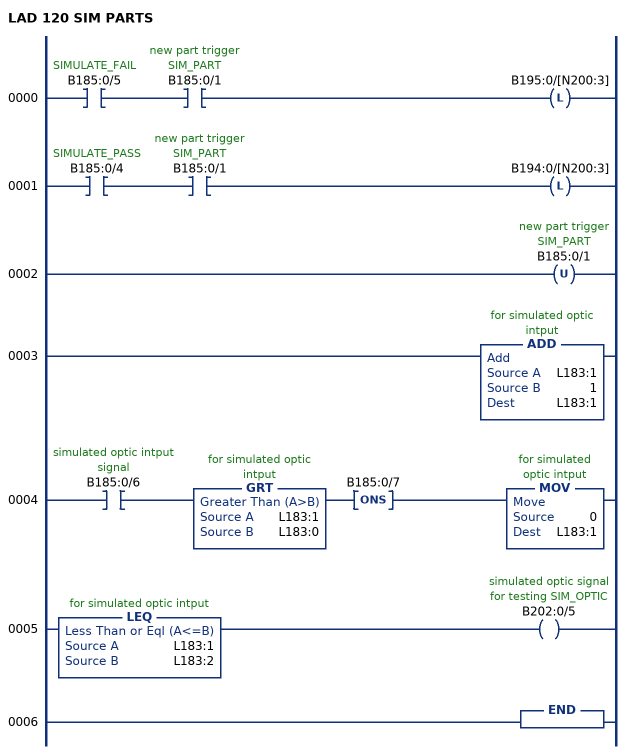
% Rung: 0 %
SOR XIC B185:0/5 XIC B185:0/1 OTL B195:0/[N200:3] EOR
%   B185:0/5  SIMULATE_FAIL %
%   B185:0/1  SIM_PART  "new part trigger" %
%   N200:3  OPT_LD_PT %
% Rung: 1 %
SOR XIC B185:0/4 XIC B185:0/1 OTL B194:0/[N200:3] EOR
%   B185:0/4  SIMULATE_PASS %
%   B185:0/1  SIM_PART  "new part trigger" %
%   N200:3  OPT_LD_PT %
% Rung: 2 %
SOR OTU B185:0/1 EOR
%   B185:0/1  SIM_PART  "new part trigger" %
% Rung: 3 %
SOR ADD L183:1 1 L183:1 EOR
%   L183:1  "for simulated optic intput" %
% Rung: 4 %
SOR XIC B185:0/6 GRT L183:1 L183:0 ONS B185:0/7 MOV 0 L183:1 EOR
%   B185:0/6  "simulated optic intput signal" %
%   L183:1  "for simulated optic intput" %
%   L183:0  "count for part data injection" %
% Rung: 5 %
SOR LEQ L183:1 L183:2 OTE B202:0/5 EOR
%   L183:1  "for simulated optic intput" %
%   L183:2  "simulated part width" %
%   B202:0/5  SIM_OPTIC  "simulated optic signal for testing" %
% Rung: 6 %
SOR END EOR

LADDER 121 "PARTDETECT"
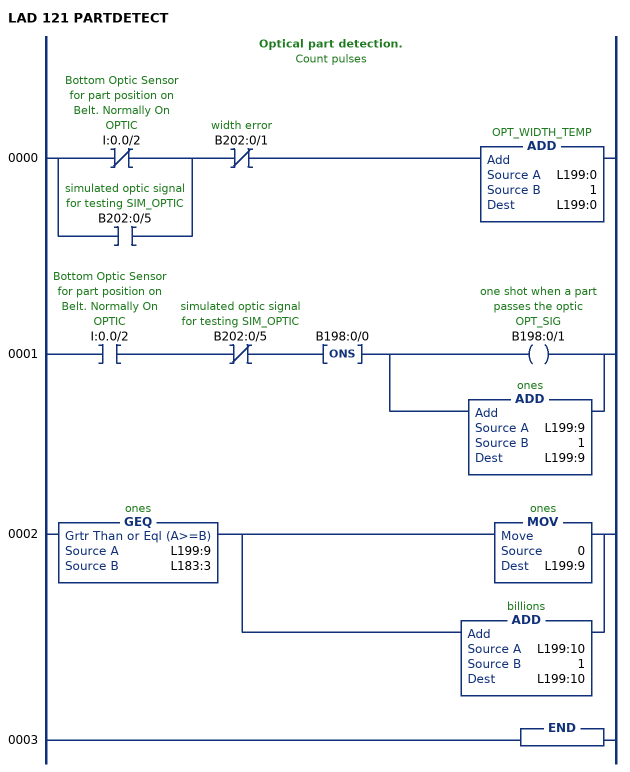
% Rung: 0 %
% TITLE: Optical part detection. %
% Count pulses %
SOR BST XIO I:0.0/2 NXB XIC B202:0/5 BND XIO B202:0/1 ADD L199:0 1 L199:0 EOR
%   I:0.0/2  OPTIC  "Bottom Optic Sensor for part position on Belt. Normally On" %
%   B202:0/5  SIM_OPTIC  "simulated optic signal for testing" %
%   B202:0/1  "width error" %
%   L199:0  OPT_WIDTH_TEMP %
% Rung: 1 %
SOR XIC I:0.0/2 XIO B202:0/5 ONS B198:0/0 BST OTE B198:0/1 NXB ADD L199:9 1 L199:9 BND EOR
%   I:0.0/2  OPTIC  "Bottom Optic Sensor for part position on Belt. Normally On" %
%   B202:0/5  SIM_OPTIC  "simulated optic signal for testing" %
%   B198:0/1  OPT_SIG  "one shot when a part passes the optic" %
%   L199:9  "ones" %
% Rung: 2 %
SOR GEQ L199:9 L183:3 BST MOV 0 L199:9 NXB ADD L199:10 1 L199:10 BND EOR
%   L199:9  "ones" %
%   L183:3  "button state" %
%   L199:10  "billions" %
% Rung: 3 %
SOR END EOR

LADDER 122 "OPTICWIDTH"
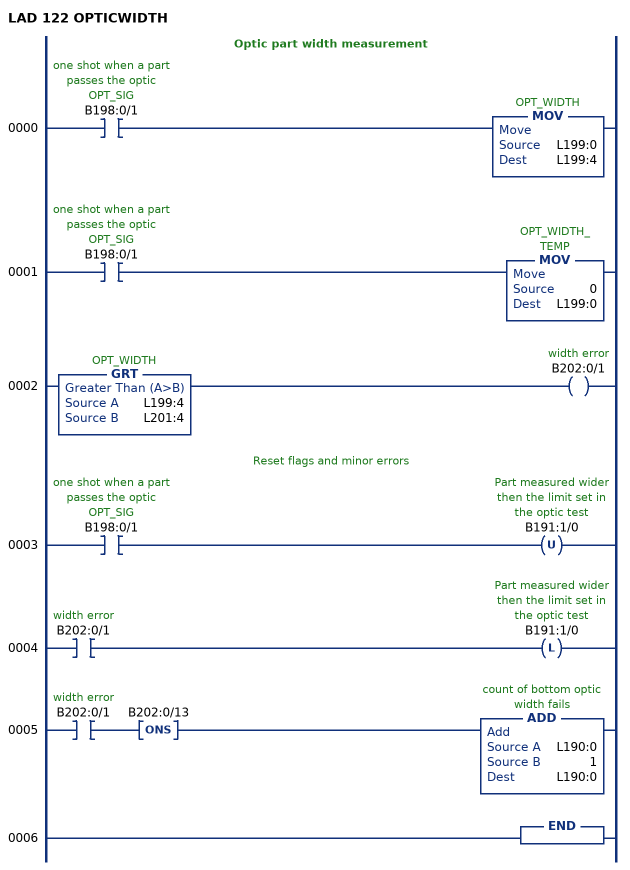
% Rung: 0 %
% TITLE: Optic part width measurement %
SOR XIC B198:0/1 MOV L199:0 L199:4 EOR
%   B198:0/1  OPT_SIG  "one shot when a part passes the optic" %
%   L199:0  OPT_WIDTH_TEMP %
%   L199:4  OPT_WIDTH %
% Rung: 1 %
SOR XIC B198:0/1 MOV 0 L199:0 EOR
%   B198:0/1  OPT_SIG  "one shot when a part passes the optic" %
%   L199:0  OPT_WIDTH_TEMP %
% Rung: 2 %
SOR GRT L199:4 L201:4 OTE B202:0/1 EOR
%   L199:4  OPT_WIDTH %
%   L201:4  MAX_WIDTH  "hmi in" %
%   B202:0/1  "width error" %
% Rung: 3 %
% Reset flags and minor errors %
SOR XIC B198:0/1 OTU B191:1/0 EOR
%   B198:0/1  OPT_SIG  "one shot when a part passes the optic" %
%   B191:1/0  "Part measured wider then the limit set in the optic test" %
% Rung: 4 %
SOR XIC B202:0/1 OTL B191:1/0 EOR
%   B202:0/1  "width error" %
%   B191:1/0  "Part measured wider then the limit set in the optic test" %
% Rung: 5 %
SOR XIC B202:0/1 ONS B202:0/13 ADD L190:0 1 L190:0 EOR
%   B202:0/1  "width error" %
%   L190:0  "count of bottom optic width fails" %
% Rung: 6 %
SOR END EOR

LADDER 123 "PART GAP"
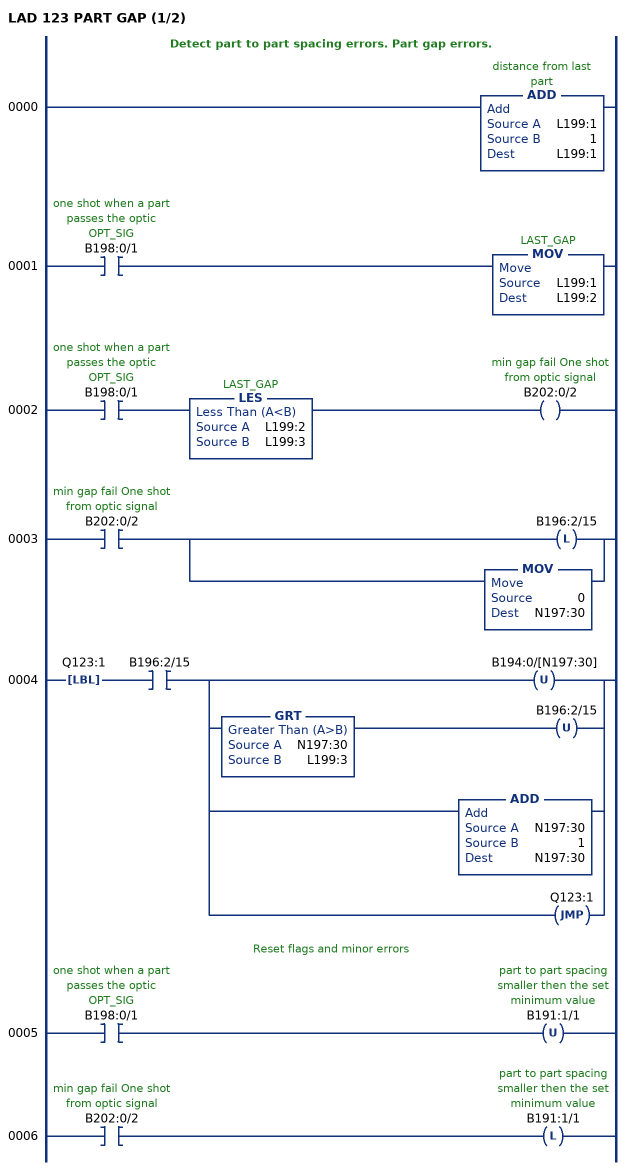
% Rung: 0 %
% TITLE: Detect part to part spacing errors. Part gap errors. %
SOR ADD L199:1 1 L199:1 EOR
%   L199:1  "distance from last part" %
% Rung: 1 %
SOR XIC B198:0/1 MOV L199:1 L199:2 EOR
%   B198:0/1  OPT_SIG  "one shot when a part passes the optic" %
%   L199:1  "distance from last part" %
%   L199:2  LAST_GAP %
% Rung: 2 %
SOR XIC B198:0/1 LES L199:2 L199:3 OTE B202:0/2 EOR
%   B198:0/1  OPT_SIG  "one shot when a part passes the optic" %
%   L199:2  LAST_GAP %
%   L199:3  MIN_WIDTH %
%   B202:0/2  "min gap fail One shot from optic signal" %
% Rung: 3 %
SOR XIC B202:0/2 BST OTL B196:2/15 NXB MOV 0 N197:30 BND EOR
%   B202:0/2  "min gap fail One shot from optic signal" %
% Rung: 4 %
SOR LBL Q123:1 XIC B196:2/15 BST OTU B194:0/[N197:30] NXB GRT N197:30 L199:3 OTU B196:2/15 NXB ADD N197:30 1 N197:30 NXB JMP Q123:1 BND EOR
%   L199:3  MIN_WIDTH %
% Rung: 5 %
% Reset flags and minor errors %
SOR XIC B198:0/1 OTU B191:1/1 EOR
%   B198:0/1  OPT_SIG  "one shot when a part passes the optic" %
%   B191:1/1  "part to part spacing smaller then the set minimum value" %
% Rung: 6 %
SOR XIC B202:0/2 OTL B191:1/1 EOR
%   B202:0/2  "min gap fail One shot from optic signal" %
%   B191:1/1  "part to part spacing smaller then the set minimum value" %

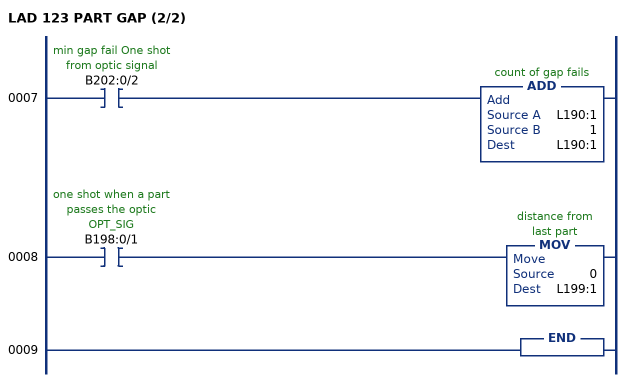
% Rung: 7 %
SOR XIC B202:0/2 ADD L190:1 1 L190:1 EOR
%   B202:0/2  "min gap fail One shot from optic signal" %
%   L190:1  "count of gap fails" %
% Rung: 8 %
SOR XIC B198:0/1 MOV 0 L199:1 EOR
%   B198:0/1  OPT_SIG  "one shot when a part passes the optic" %
%   L199:1  "distance from last part" %
% Rung: 9 %
SOR END EOR

LADDER 125 "OPTIC"
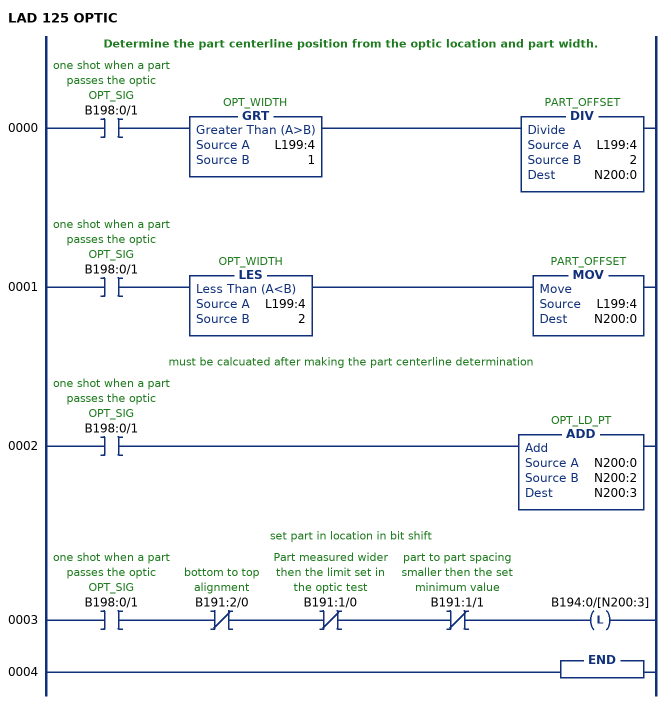
% Rung: 0 %
% TITLE: Determine the part centerline position from the optic location and part width. %
SOR XIC B198:0/1 GRT L199:4 1 DIV L199:4 2 N200:0 EOR
%   B198:0/1  OPT_SIG  "one shot when a part passes the optic" %
%   L199:4  OPT_WIDTH %
%   N200:0  PART_OFFSET %
% Rung: 1 %
SOR XIC B198:0/1 LES L199:4 2 MOV L199:4 N200:0 EOR
%   B198:0/1  OPT_SIG  "one shot when a part passes the optic" %
%   L199:4  OPT_WIDTH %
%   N200:0  PART_OFFSET %
% Rung: 2 %
% must be calcuated after making the part centerline determination %
SOR XIC B198:0/1 ADD N200:0 N200:2 N200:3 EOR
%   B198:0/1  OPT_SIG  "one shot when a part passes the optic" %
%   N200:0  PART_OFFSET %
%   N200:2  OPTIC_LOC %
%   N200:3  OPT_LD_PT %
% Rung: 3 %
% set part in location in bit shift %
SOR XIC B198:0/1 XIO B191:2/0 XIO B191:1/0 XIO B191:1/1 OTL B194:0/[N200:3] EOR
%   B198:0/1  OPT_SIG  "one shot when a part passes the optic" %
%   B191:2/0  "bottom to top alignment" %
%   B191:1/0  "Part measured wider then the limit set in the optic test" %
%   B191:1/1  "part to part spacing smaller then the set minimum value" %
%   N200:3  OPT_LD_PT %
% Rung: 4 %
SOR END EOR

LADDER 130 "INS 1 TRIG"
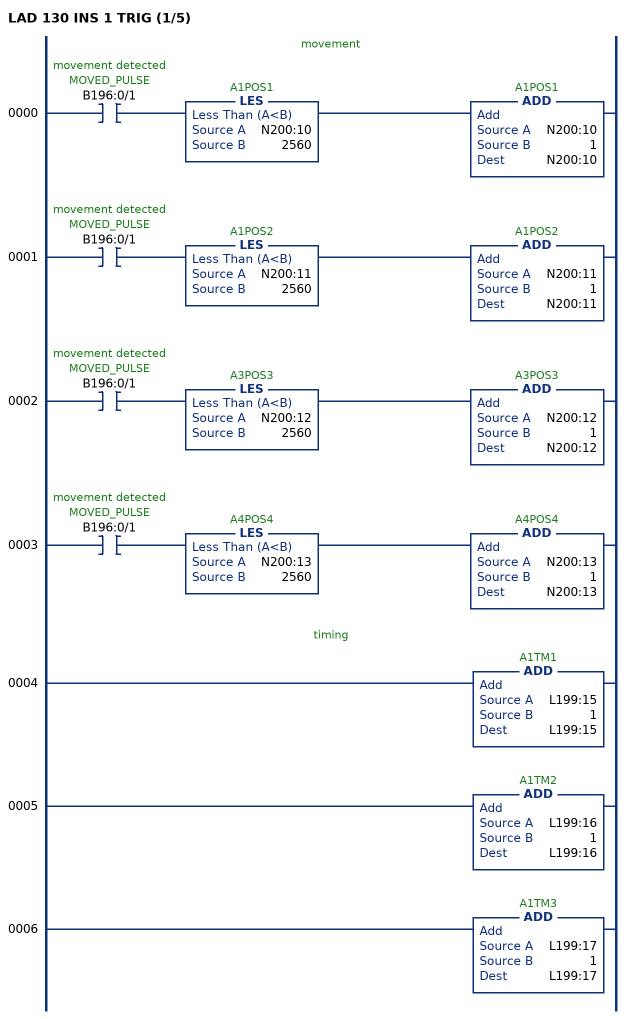
% Rung: 0 %
% movement %
SOR XIC B196:0/1 LES N200:10 2560 ADD N200:10 1 N200:10 EOR
%   B196:0/1  MOVED_PULSE  "movement detected" %
%   N200:10  A1POS1 %
% Rung: 1 %
SOR XIC B196:0/1 LES N200:11 2560 ADD N200:11 1 N200:11 EOR
%   B196:0/1  MOVED_PULSE  "movement detected" %
%   N200:11  A1POS2 %
% Rung: 2 %
SOR XIC B196:0/1 LES N200:12 2560 ADD N200:12 1 N200:12 EOR
%   B196:0/1  MOVED_PULSE  "movement detected" %
%   N200:12  A3POS3 %
% Rung: 3 %
SOR XIC B196:0/1 LES N200:13 2560 ADD N200:13 1 N200:13 EOR
%   B196:0/1  MOVED_PULSE  "movement detected" %
%   N200:13  A4POS4 %
% Rung: 4 %
% timing %
SOR ADD L199:15 1 L199:15 EOR
%   L199:15  A1TM1 %
% Rung: 5 %
SOR ADD L199:16 1 L199:16 EOR
%   L199:16  A1TM2 %
% Rung: 6 %
SOR ADD L199:17 1 L199:17 EOR
%   L199:17  A1TM3 %

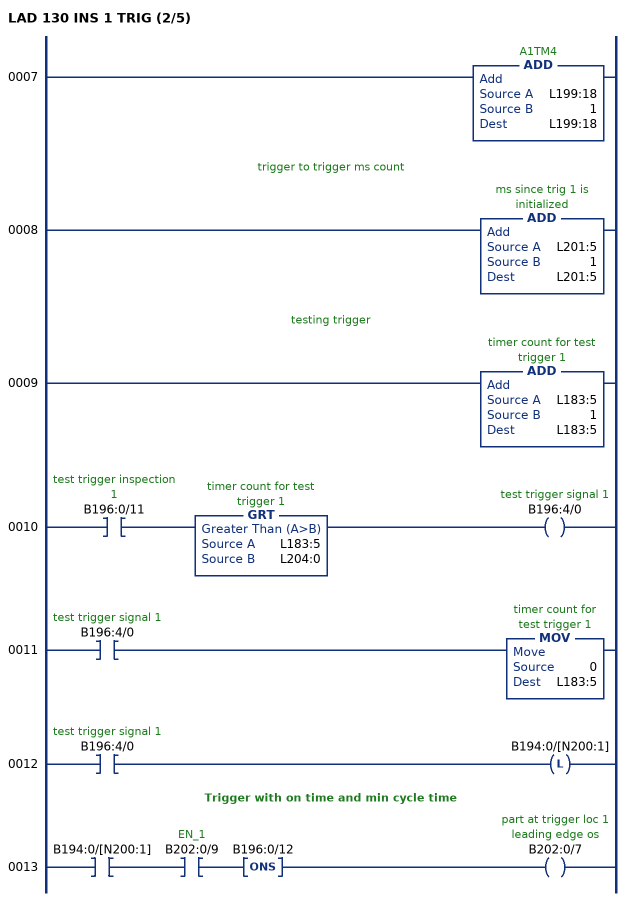
% Rung: 7 %
SOR ADD L199:18 1 L199:18 EOR
%   L199:18  A1TM4 %
% Rung: 8 %
% trigger to trigger ms count %
SOR ADD L201:5 1 L201:5 EOR
%   L201:5  "ms since trig 1 is initialized" %
% Rung: 9 %
% testing trigger %
SOR ADD L183:5 1 L183:5 EOR
%   L183:5  "timer count for test trigger 1" %
% Rung: 10 %
SOR XIC B196:0/11 GRT L183:5 L204:0 OTE B196:4/0 EOR
%   B196:0/11  "test trigger inspection 1" %
%   L183:5  "timer count for test trigger 1" %
%   B196:4/0  "test trigger signal 1" %
% Rung: 11 %
SOR XIC B196:4/0 MOV 0 L183:5 EOR
%   B196:4/0  "test trigger signal 1" %
%   L183:5  "timer count for test trigger 1" %
% Rung: 12 %
SOR XIC B196:4/0 OTL B194:0/[N200:1] EOR
%   B196:4/0  "test trigger signal 1" %
%   N200:1  INS_1_TRIG_LOC %
% Rung: 13 %
% TITLE: Trigger with on time and min cycle time %
SOR XIC B194:0/[N200:1] XIC B202:0/9 ONS B196:0/12 OTE B202:0/7 EOR
%   N200:1  INS_1_TRIG_LOC %
%   B202:0/9  EN_1 %
%   B202:0/7  "part at trigger loc 1 leading edge os" %

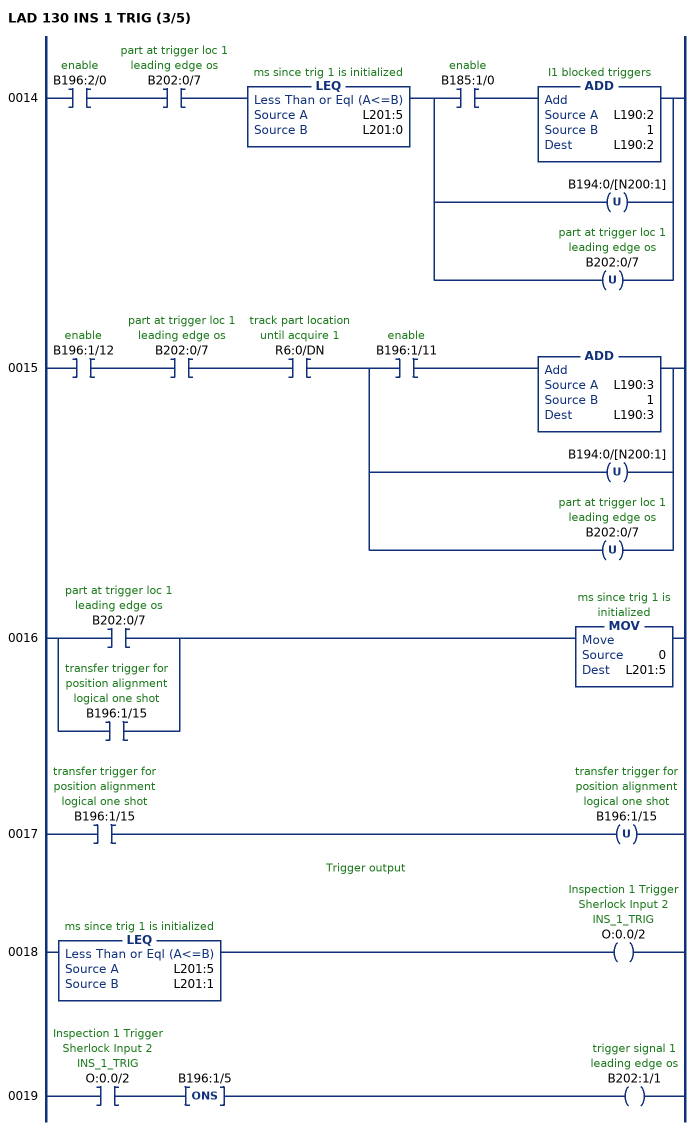
% Rung: 14 %
SOR XIC B196:2/0 XIC B202:0/7 LEQ L201:5 L201:0 BST XIC B185:1/0 ADD L190:2 1 L190:2 NXB OTU B194:0/[N200:1] NXB OTU B202:0/7 BND EOR
%   B196:2/0  "enable" %
%   B202:0/7  "part at trigger loc 1 leading edge os" %
%   L201:5  "ms since trig 1 is initialized" %
%   L201:0  CAM_1_MIN_CYCLE_TIME %
%   B185:1/0  "enable" %
%   L190:2  "I1 blocked triggers" %
%   N200:1  INS_1_TRIG_LOC %
% Rung: 15 %
SOR XIC B196:1/12 XIC B202:0/7 XIC R6:0/DN BST XIC B196:1/11 ADD L190:3 1 L190:3 NXB OTU B194:0/[N200:1] NXB OTU B202:0/7 BND EOR
%   B196:1/12  "enable" %
%   B202:0/7  "part at trigger loc 1 leading edge os" %
%   R6:0  "track part location until acquire 1" %
%   B196:1/11  "enable" %
%   N200:1  INS_1_TRIG_LOC %
% Rung: 16 %
SOR BST XIC B202:0/7 NXB XIC B196:1/15 BND MOV 0 L201:5 EOR
%   B202:0/7  "part at trigger loc 1 leading edge os" %
%   B196:1/15  "transfer trigger for position alignment logical one shot" %
%   L201:5  "ms since trig 1 is initialized" %
% Rung: 17 %
SOR XIC B196:1/15 OTU B196:1/15 EOR
%   B196:1/15  "transfer trigger for position alignment logical one shot" %
% Rung: 18 %
% Trigger output %
SOR LEQ L201:5 L201:1 OTE O:0.0/2 EOR
%   L201:5  "ms since trig 1 is initialized" %
%   L201:1  CAM_1_TRIG_TIME  "out time" %
%   O:0.0/2  INS_1_TRIG  "Inspection 1 Trigger Sherlock Input 2" %
% Rung: 19 %
SOR XIC O:0.0/2 ONS B196:1/5 OTE B202:1/1 EOR
%   O:0.0/2  INS_1_TRIG  "Inspection 1 Trigger Sherlock Input 2" %
%   B202:1/1  "trigger signal 1 leading edge os" %

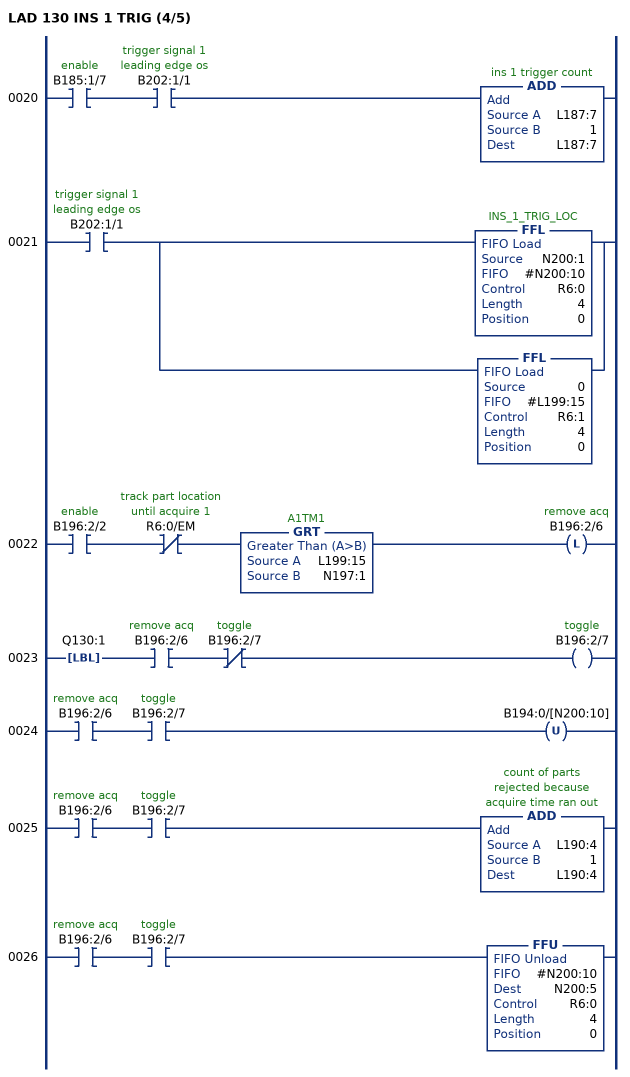
% Rung: 20 %
SOR XIC B185:1/7 XIC B202:1/1 ADD L187:7 1 L187:7 EOR
%   B185:1/7  "enable" %
%   B202:1/1  "trigger signal 1 leading edge os" %
%   L187:7  "ins 1 trigger count" %
% Rung: 21 %
SOR XIC B202:1/1 BST FFL N200:1 #N200:10 R6:0 4 0 NXB FFL 0 #L199:15 R6:1 4 0 BND EOR
%   B202:1/1  "trigger signal 1 leading edge os" %
%   N200:1  INS_1_TRIG_LOC %
%   N200:10  A1POS1 %
%   R6:0  "track part location until acquire 1" %
%   L199:15  A1TM1 %
%   R6:1  "track acquire time 1" %
% Rung: 22 %
SOR XIC B196:2/2 XIO R6:0/EM GRT L199:15 N197:1 OTL B196:2/6 EOR
%   B196:2/2  "enable" %
%   R6:0  "track part location until acquire 1" %
%   L199:15  A1TM1 %
%   N197:1  "maximim acquire time 1" %
%   B196:2/6  "remove acq" %
% Rung: 23 %
SOR LBL Q130:1 XIC B196:2/6 XIO B196:2/7 OTE B196:2/7 EOR
%   B196:2/6  "remove acq" %
%   B196:2/7  "toggle" %
% Rung: 24 %
SOR XIC B196:2/6 XIC B196:2/7 OTU B194:0/[N200:10] EOR
%   B196:2/6  "remove acq" %
%   B196:2/7  "toggle" %
%   N200:10  A1POS1 %
% Rung: 25 %
SOR XIC B196:2/6 XIC B196:2/7 ADD L190:4 1 L190:4 EOR
%   B196:2/6  "remove acq" %
%   B196:2/7  "toggle" %
%   L190:4  "count of parts rejected because acquire time ran out" %
% Rung: 26 %
SOR XIC B196:2/6 XIC B196:2/7 FFU #N200:10 N200:5 R6:0 4 0 EOR
%   B196:2/6  "remove acq" %
%   B196:2/7  "toggle" %
%   N200:10  A1POS1 %
%   R6:0  "track part location until acquire 1" %

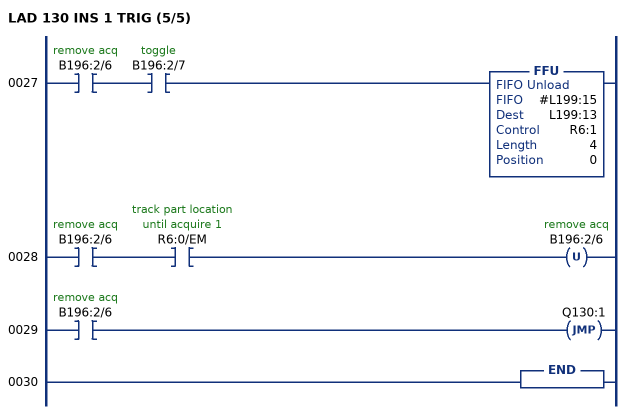
% Rung: 27 %
SOR XIC B196:2/6 XIC B196:2/7 FFU #L199:15 L199:13 R6:1 4 0 EOR
%   B196:2/6  "remove acq" %
%   B196:2/7  "toggle" %
%   L199:15  A1TM1 %
%   R6:1  "track acquire time 1" %
% Rung: 28 %
SOR XIC B196:2/6 XIC R6:0/EM OTU B196:2/6 EOR
%   B196:2/6  "remove acq" %
%   R6:0  "track part location until acquire 1" %
% Rung: 29 %
SOR XIC B196:2/6 JMP Q130:1 EOR
%   B196:2/6  "remove acq" %
% Rung: 30 %
SOR END EOR

LADDER 131 "INS 1 RSLT"
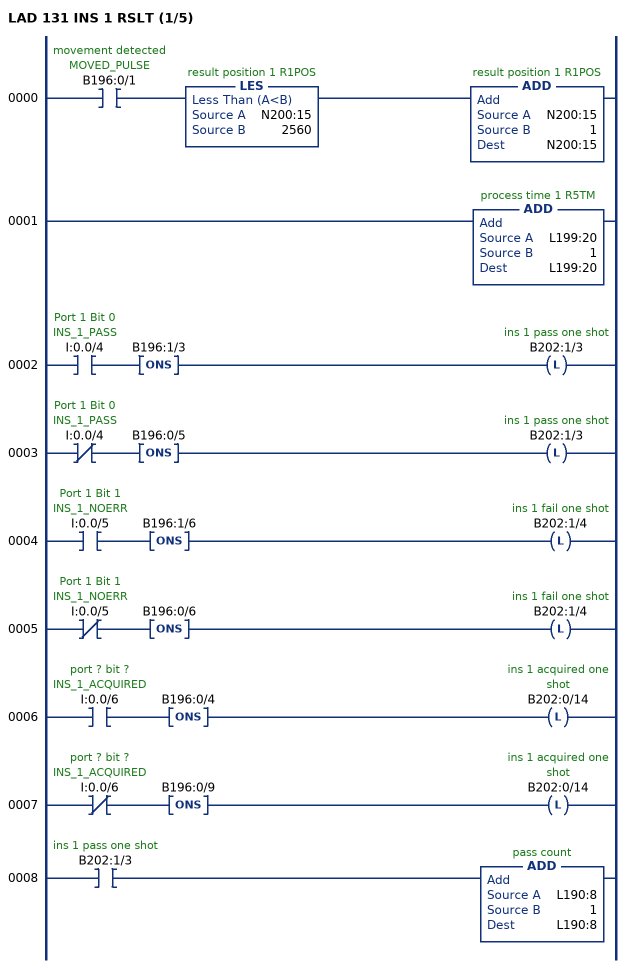
% Rung: 0 %
SOR XIC B196:0/1 LES N200:15 2560 ADD N200:15 1 N200:15 EOR
%   B196:0/1  MOVED_PULSE  "movement detected" %
%   N200:15  R1POS  "result position 1" %
% Rung: 1 %
SOR ADD L199:20 1 L199:20 EOR
%   L199:20  R5TM  "process time 1" %
% Rung: 2 %
SOR XIC I:0.0/4 ONS B196:1/3 OTL B202:1/3 EOR
%   I:0.0/4  INS_1_PASS  "Port 1 Bit 0" %
%   B202:1/3  "ins 1 pass one shot" %
% Rung: 3 %
SOR XIO I:0.0/4 ONS B196:0/5 OTL B202:1/3 EOR
%   I:0.0/4  INS_1_PASS  "Port 1 Bit 0" %
%   B202:1/3  "ins 1 pass one shot" %
% Rung: 4 %
SOR XIC I:0.0/5 ONS B196:1/6 OTL B202:1/4 EOR
%   I:0.0/5  INS_1_NOERR  "Port 1 Bit 1" %
%   B202:1/4  "ins 1 fail one shot" %
% Rung: 5 %
SOR XIO I:0.0/5 ONS B196:0/6 OTL B202:1/4 EOR
%   I:0.0/5  INS_1_NOERR  "Port 1 Bit 1" %
%   B202:1/4  "ins 1 fail one shot" %
% Rung: 6 %
SOR XIC I:0.0/6 ONS B196:0/4 OTL B202:0/14 EOR
%   I:0.0/6  INS_1_ACQUIRED  "port ? bit ?" %
%   B202:0/14  "ins 1 acquired one shot" %
% Rung: 7 %
SOR XIO I:0.0/6 ONS B196:0/9 OTL B202:0/14 EOR
%   I:0.0/6  INS_1_ACQUIRED  "port ? bit ?" %
%   B202:0/14  "ins 1 acquired one shot" %
% Rung: 8 %
SOR XIC B202:1/3 ADD L190:8 1 L190:8 EOR
%   B202:1/3  "ins 1 pass one shot" %
%   L190:8  "pass count" %

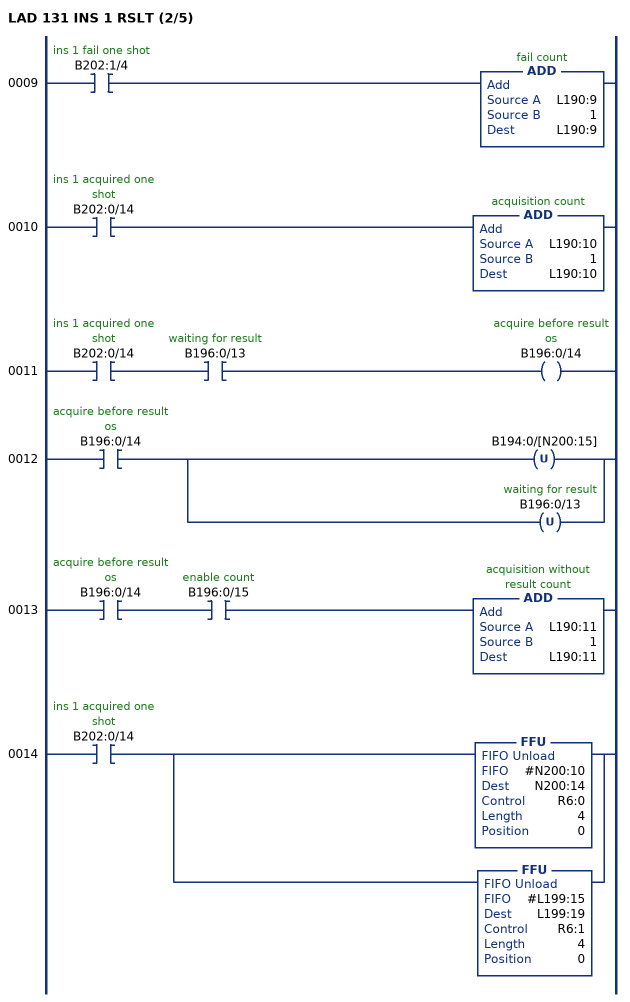
% Rung: 9 %
SOR XIC B202:1/4 ADD L190:9 1 L190:9 EOR
%   B202:1/4  "ins 1 fail one shot" %
%   L190:9  "fail count" %
% Rung: 10 %
SOR XIC B202:0/14 ADD L190:10 1 L190:10 EOR
%   B202:0/14  "ins 1 acquired one shot" %
%   L190:10  "acquisition count" %
% Rung: 11 %
SOR XIC B202:0/14 XIC B196:0/13 OTE B196:0/14 EOR
%   B202:0/14  "ins 1 acquired one shot" %
%   B196:0/13  "waiting for result" %
%   B196:0/14  "acquire before result os" %
% Rung: 12 %
SOR XIC B196:0/14 BST OTU B194:0/[N200:15] NXB OTU B196:0/13 BND EOR
%   B196:0/14  "acquire before result os" %
%   N200:15  R1POS  "result position 1" %
%   B196:0/13  "waiting for result" %
% Rung: 13 %
SOR XIC B196:0/14 XIC B196:0/15 ADD L190:11 1 L190:11 EOR
%   B196:0/14  "acquire before result os" %
%   B196:0/15  "enable count" %
%   L190:11  "acquisition without result count" %
% Rung: 14 %
SOR XIC B202:0/14 BST FFU #N200:10 N200:14 R6:0 4 0 NXB FFU #L199:15 L199:19 R6:1 4 0 BND EOR
%   B202:0/14  "ins 1 acquired one shot" %
%   N200:10  A1POS1 %
%   R6:0  "track part location until acquire 1" %
%   L199:15  A1TM1 %
%   R6:1  "track acquire time 1" %

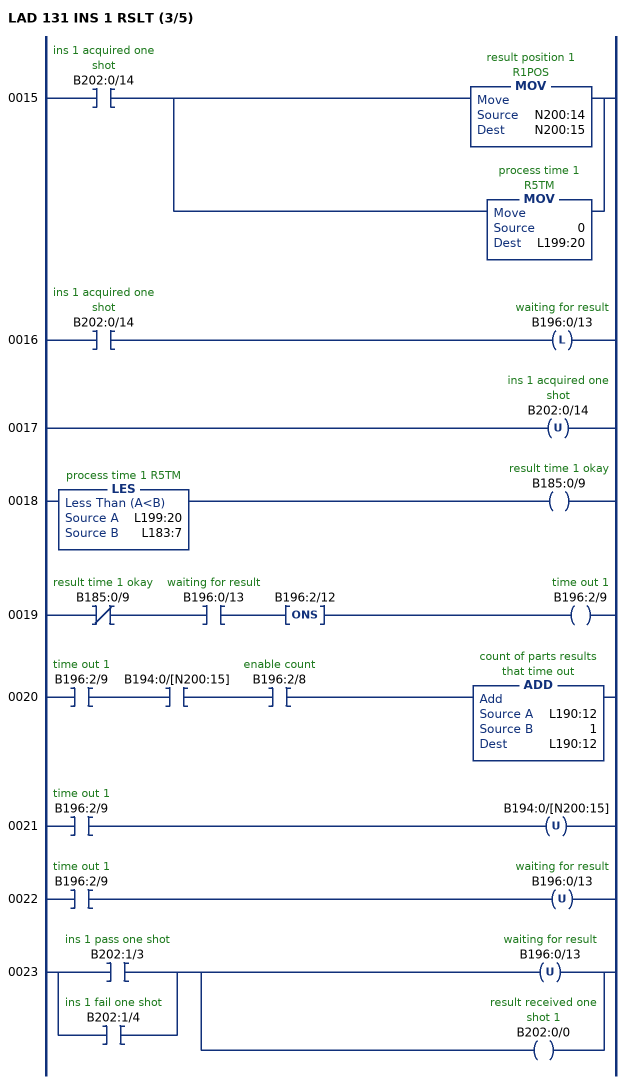
% Rung: 15 %
SOR XIC B202:0/14 BST MOV N200:14 N200:15 NXB MOV 0 L199:20 BND EOR
%   B202:0/14  "ins 1 acquired one shot" %
%   N200:15  R1POS  "result position 1" %
%   L199:20  R5TM  "process time 1" %
% Rung: 16 %
SOR XIC B202:0/14 OTL B196:0/13 EOR
%   B202:0/14  "ins 1 acquired one shot" %
%   B196:0/13  "waiting for result" %
% Rung: 17 %
SOR OTU B202:0/14 EOR
%   B202:0/14  "ins 1 acquired one shot" %
% Rung: 18 %
SOR LES L199:20 L183:7 OTE B185:0/9 EOR
%   L199:20  R5TM  "process time 1" %
%   L183:7  "max process time 1" %
%   B185:0/9  "result time 1 okay" %
% Rung: 19 %
SOR XIO B185:0/9 XIC B196:0/13 ONS B196:2/12 OTE B196:2/9 EOR
%   B185:0/9  "result time 1 okay" %
%   B196:0/13  "waiting for result" %
%   B196:2/9  "time out 1" %
% Rung: 20 %
SOR XIC B196:2/9 XIC B194:0/[N200:15] XIC B196:2/8 ADD L190:12 1 L190:12 EOR
%   B196:2/9  "time out 1" %
%   N200:15  R1POS  "result position 1" %
%   B196:2/8  "enable count" %
%   L190:12  "count of parts results that time out" %
% Rung: 21 %
SOR XIC B196:2/9 OTU B194:0/[N200:15] EOR
%   B196:2/9  "time out 1" %
%   N200:15  R1POS  "result position 1" %
% Rung: 22 %
SOR XIC B196:2/9 OTU B196:0/13 EOR
%   B196:2/9  "time out 1" %
%   B196:0/13  "waiting for result" %
% Rung: 23 %
SOR BST XIC B202:1/3 NXB XIC B202:1/4 BND BST OTU B196:0/13 NXB OTE B202:0/0 BND EOR
%   B202:1/3  "ins 1 pass one shot" %
%   B202:1/4  "ins 1 fail one shot" %
%   B196:0/13  "waiting for result" %
%   B202:0/0  "result received one shot 1" %

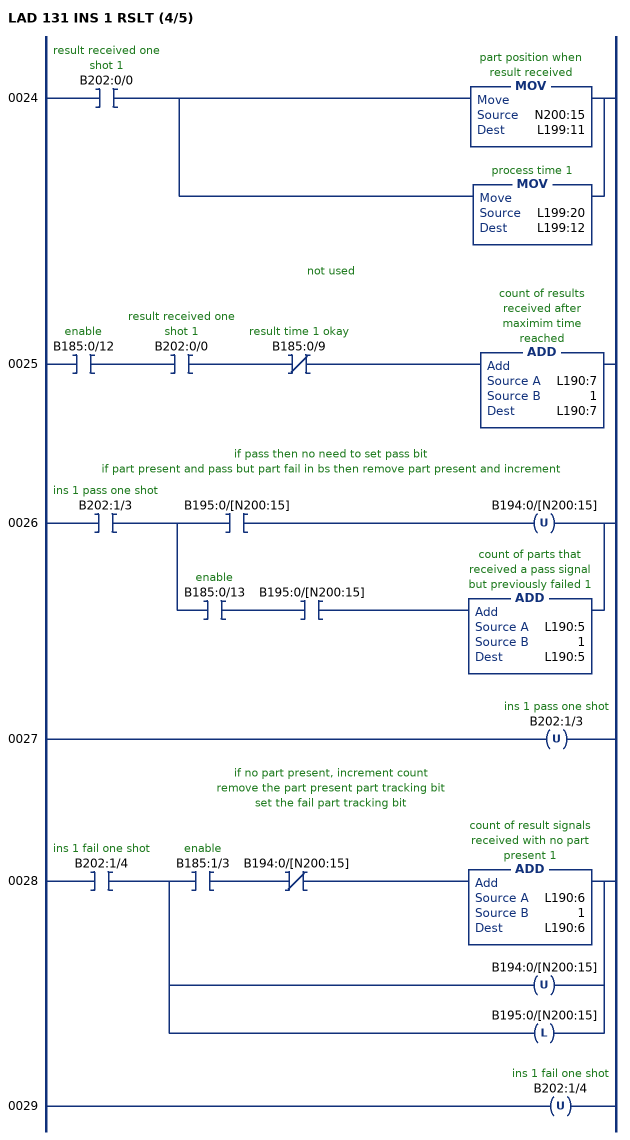
% Rung: 24 %
SOR XIC B202:0/0 BST MOV N200:15 L199:11 NXB MOV L199:20 L199:12 BND EOR
%   B202:0/0  "result received one shot 1" %
%   N200:15  R1POS  "result position 1" %
%   L199:11  "part position when result received" %
%   L199:20  R5TM  "process time 1" %
%   L199:12  "process time 1" %
% Rung: 25 %
% not used %
SOR XIC B185:0/12 XIC B202:0/0 XIO B185:0/9 ADD L190:7 1 L190:7 EOR
%   B185:0/12  "enable" %
%   B202:0/0  "result received one shot 1" %
%   B185:0/9  "result time 1 okay" %
%   L190:7  "count of results received after maximim time reached" %
% Rung: 26 %
% if pass then no need to set pass bit
% if part present and pass but part fail in bs then remove part present and increment %
SOR XIC B202:1/3 BST XIC B195:0/[N200:15] OTU B194:0/[N200:15] NXB XIC B185:0/13 XIC B195:0/[N200:15] ADD L190:5 1 L190:5 BND EOR
%   B202:1/3  "ins 1 pass one shot" %
%   N200:15  R1POS  "result position 1" %
%   B185:0/13  "enable" %
%   L190:5  "count of parts that received a pass signal but previously failed 1" %
% Rung: 27 %
SOR OTU B202:1/3 EOR
%   B202:1/3  "ins 1 pass one shot" %
% Rung: 28 %
% if no part present, increment count
% remove the part present part tracking bit
% set the fail part tracking bit %
SOR XIC B202:1/4 BST XIC B185:1/3 XIO B194:0/[N200:15] ADD L190:6 1 L190:6 NXB OTU B194:0/[N200:15] NXB OTL B195:0/[N200:15] BND EOR
%   B202:1/4  "ins 1 fail one shot" %
%   B185:1/3  "enable" %
%   N200:15  R1POS  "result position 1" %
%   L190:6  "count of result signals received with no part present 1" %
% Rung: 29 %
SOR OTU B202:1/4 EOR
%   B202:1/4  "ins 1 fail one shot" %

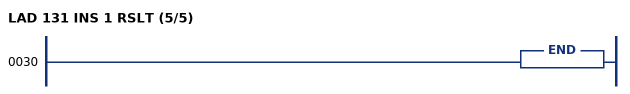
% Rung: 30 %
SOR END EOR

LADDER 150 "DEF HEAD"    % remove me %
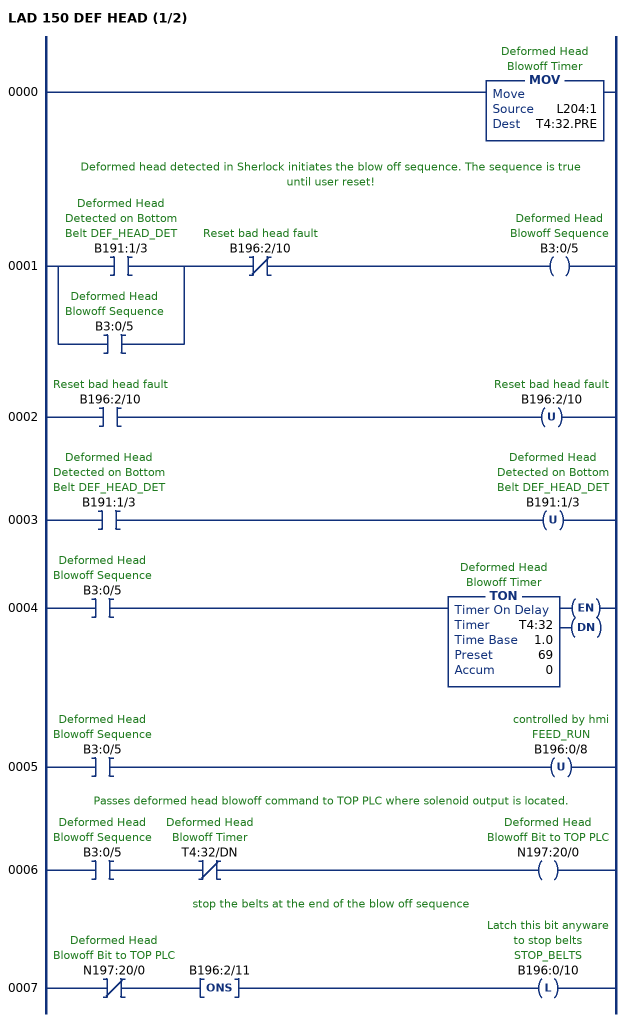
% Rung: 0 %
SOR MOV L204:1 T4:32.PRE EOR
%   L204:1  BELT_STOP_VALUE  "the value that when the belt tic reaches will cause the belt to stop" %
%   T4:32  "Deformed Head Blowoff Timer" %
% Rung: 1 %
% Deformed head detected in Sherlock initiates the blow off sequence. The sequence is true until user reset! %
SOR BST XIC B191:1/3 NXB XIC B3:0/5 BND XIO B196:2/10 OTE B3:0/5 EOR
%   B191:1/3  DEF_HEAD_DET  "Deformed Head Detected on Bottom Belt" %
%   B3:0/5  "Deformed Head Blowoff Sequence" %
%   B196:2/10  "Reset bad head fault" %
% Rung: 2 %
SOR XIC B196:2/10 OTU B196:2/10 EOR
%   B196:2/10  "Reset bad head fault" %
% Rung: 3 %
SOR XIC B191:1/3 OTU B191:1/3 EOR
%   B191:1/3  DEF_HEAD_DET  "Deformed Head Detected on Bottom Belt" %
% Rung: 4 %
SOR XIC B3:0/5 TON T4:32 1.0 69 0 EOR
%   B3:0/5  "Deformed Head Blowoff Sequence" %
%   T4:32  "Deformed Head Blowoff Timer" %
% Rung: 5 %
SOR XIC B3:0/5 OTU B196:0/8 EOR
%   B3:0/5  "Deformed Head Blowoff Sequence" %
%   B196:0/8  FEED_RUN  "controlled by hmi" %
% Rung: 6 %
% Passes deformed head blowoff command to TOP PLC where solenoid output is located. %
SOR XIC B3:0/5 XIO T4:32/DN OTE N197:20/0 EOR
%   B3:0/5  "Deformed Head Blowoff Sequence" %
%   T4:32  "Deformed Head Blowoff Timer" %
%   N197:20/0  "Deformed Head Blowoff Bit to TOP PLC" %
% Rung: 7 %
% stop the belts at the end of the blow off sequence %
SOR XIO N197:20/0 ONS B196:2/11 OTL B196:0/10 EOR
%   N197:20/0  "Deformed Head Blowoff Bit to TOP PLC" %
%   B196:0/10  STOP_BELTS  "Latch this bit anyware to stop belts" %

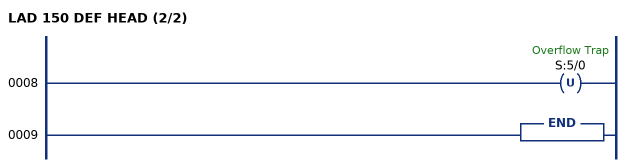
% Rung: 8 %
SOR OTU S:5/0 EOR
%   S:5/0  "Overflow Trap" %
% Rung: 9 %
SOR END EOR

LADDER 170 "XFER OUT"
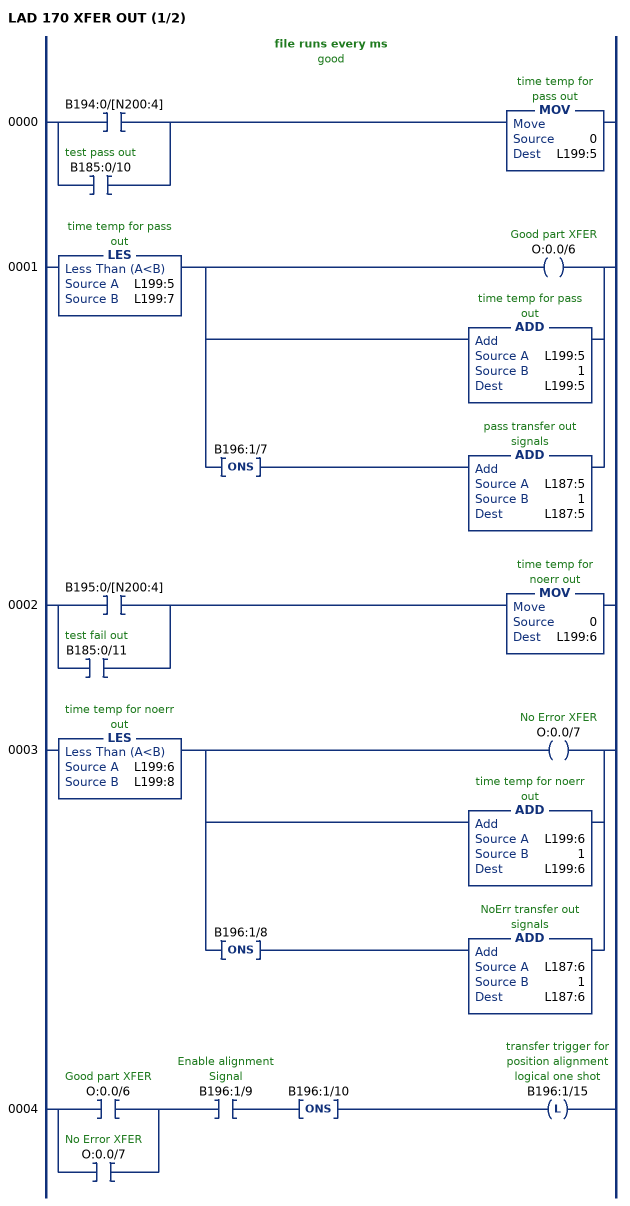
% Rung: 0 %
% TITLE: file runs every ms %
% good %
SOR BST XIC B194:0/[N200:4] NXB XIC B185:0/10 BND MOV 0 L199:5 EOR
%   N200:4  XFER_OUT  "The location to send the data out to the other inspection" %
%   B185:0/10  "test pass out" %
%   L199:5  "time temp for pass out" %
% Rung: 1 %
SOR LES L199:5 L199:7 BST OTE O:0.0/6 NXB ADD L199:5 1 L199:5 NXB ONS B196:1/7 ADD L187:5 1 L187:5 BND EOR
%   L199:5  "time temp for pass out" %
%   O:0.0/6  "Good part XFER" %
%   L187:5  "pass transfer out signals" %
% Rung: 2 %
SOR BST XIC B195:0/[N200:4] NXB XIC B185:0/11 BND MOV 0 L199:6 EOR
%   N200:4  XFER_OUT  "The location to send the data out to the other inspection" %
%   B185:0/11  "test fail out" %
%   L199:6  "time temp for noerr out" %
% Rung: 3 %
SOR LES L199:6 L199:8 BST OTE O:0.0/7 NXB ADD L199:6 1 L199:6 NXB ONS B196:1/8 ADD L187:6 1 L187:6 BND EOR
%   L199:6  "time temp for noerr out" %
%   O:0.0/7  "No Error XFER" %
%   L187:6  "NoErr transfer out signals" %
% Rung: 4 %
SOR BST XIC O:0.0/6 NXB XIC O:0.0/7 BND XIC B196:1/9 ONS B196:1/10 OTL B196:1/15 EOR
%   O:0.0/6  "Good part XFER" %
%   O:0.0/7  "No Error XFER" %
%   B196:1/9  "Enable alignment Signal" %
%   B196:1/15  "transfer trigger for position alignment logical one shot" %

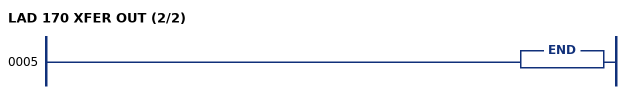
% Rung: 5 %
SOR END EOR

OTHER DOCUMENTED ADDRESSES
  100000L  
  B3:0/1  FEED_STOP  "Turn off feed"
  B3:0/2  HMI_BOX_TOG  "HMI Boxing Enable"
  B3:0/3  CONVEYORS_ENABLED  "Belt Enabled"
  B3:0/4  BYPASS_BOX_SIGNAL  "Used in HMI as memory bit. Do not write to this bit."
  B3:0/6  STL_BOT  "Bot conveyor stall detected"
  B3:0/7  "boxer backed up setter"
  B3:0/9  "bottom sudo part pulse"
  B3:0/10  "bottom belt bit shift toggle bit"
  B3:0/11  "bypass"
  B3:0/13  "bypassor"
  B3:0/15  EAT  "Enable alignment trigger"
  B3:1/0  "Reserved For Shift Registers"
  B3:1/1  "bypassor"
  B3:1/4  "bypass air fault"
  B3:1/5  OK_TO_RUN  "No safty or power issue, doesn't include high level user faults."
  B3:1/6  A_PART  "a part triggered the top optic"
  B3:1/7  "blow to chute timer run"
  B3:1/10  "Reset Box Count One Shot Transfer"
  B3:1/11  WAIT_BOX  "Packaging Conveyor Waiting For Box"
  B3:1/12  "Transfer bottom pass result from end of bottom conveyor"
  B3:1/13  "one shot"
  B3:1/14  RESET_FLT
  B3:2  FLT_ARAY  "Fault Bits Array"
  B3:2/0  CNT_SENR_FLT  "FAULT Good Part Sensor Blocked"
  B3:2/1  "FAULT Conveyor Jammed TOP_CONVEY_FLT"
  B3:2/2  "I2_CON_FAILS_FLT"
  B3:2/3  DN_TRACK_SENSOR_FLT  "FAULT Feeder Track Sensor Blocked"
  B3:2/4  BOX_JAM_FLT  "FAULT Box stuck at boxing conveyor discharge"
  B3:2/5  BOX_BACKUP_FLT  "Box Discharge Backed Up"
  B3:2/6  "FAULT Conveyor Jammed BOT_CONVEY_FLT"
  B3:2/7  AIR_FLT  "FAULT Air Pressure Low"
  B3:2/8  "I3_CON_FAILS_FLT"
  B3:2/9  "I1_CON_FAILS_FLT"
  B3:2/10  "TOP OPTIC CON FAILS FLT"
  B3:2/11  "BOT OPTIC CON FAILS FLT"
  B3:2/12  "Rate Drop Fault Possible Feed Jam"
  B3:2/13  "Fail Percent High"
  B3:2/14  FLT_BULK_CT_REACHED
  B3:3/0  "one shto"
  B3:3/1  "bypassor"
  B3:3/2  "bypassor"
  B3:3/3  "one shot"
  B3:3/4  FAULT  "FAULT Any Fault Active"
  B3:3/5  "bypassor"
  B3:3/6  "one shot"
  B3:3/7  "top trigger oneshot"
  B3:3/8  "one shot"
  B3:3/9  "bypassor"
  B3:3/10  "bypassor"
  B3:3/12  "bottom trigger oneshot"
  B3:3/13  "extra trigger 1"
  B3:3/14  1_EN
  B3:3/15  "extra trigger 2"
  B3:4/0  "custom box count reached"
  B3:4/1  2_EN
  B3:4/2  "extra trigger 3"
  B3:4/3  3_EN
  B3:4/5  "alignment trigger for top optic"
  B3:4/6  I2_TRIG_TM_OK
  B3:4/8  "Bulk count reached"
  B3:4/9  BULK_BOXING_SELECTED
  B3:4/10  CUST_BOXING_SELECTED
  B3:4/11  "one shot"
  B3:4/12  FEED_ENABLE  "Feeder Enable Bit"
  B3:4/13  STL_TOP  "Top conveyor stall detected"
  B3:4/14  "transfer timer run to next rung"
  B3:4/15  "internal or customer selected chute door control"
  B3:5/0  "one shot"
  B3:5/1  TEST_I2
  B3:5/2  STOP_CONVEYORS  "Turns off the conveyors"
  B3:5/3  TEST_I3
  B3:5/4  I2_PASS_ZONE
  B3:5/5  "bypasser"
  B3:5/7  STACK_LIGHT  "Aulternate Stack Light Operation"
  B3:5/9  LPART  "a part triggered the bottom optic or the downtrack optic"
  B3:5/11  OUR_BOXING_SELECTED  "boxing system connected and selected"
  B3:5/12  I3_PASS_ZONE
  B3:5/13  "bot result toggle"
  B3:5/15  NO_PARTS  "no parts for 60 seconds"
  B3:6/0  "good part from bottom belt at top optic position"
  B3:6/1  "top part present One Shot trailing edge"
  B3:6/2  "clear belt"
  B3:6/4  "one shot"
  B3:6/5  "bottom top camra pass zone"
  B3:6/6  "one shot"
  B3:6/7  EI3_OLD  "Enable Inspection 3"
  B3:6/8  "box count reached"
  B3:6/9  CONV_ON  "both conveyors enabled"
  B3:6/10  "Bypass un-needed code untill completed !!!!!!!!!!!!!!!!"
  B3:6/11  "bypass"
  B3:6/13  "part triped sensor w/o air blast"
  B3:6/15  "nothing"
  B3:7/0  "Start Blow One Shot Transfer"
  B3:7/2  "bypass"
  B3:7/3  "one shot"
  B3:7/4  "Side trigger oneshot"
  B3:7/5  "extra bypass"
  B3:7/6  CHUTE_OPT  "Stable chute optic output"
  B3:7/7  "one shot"
  B3:7/8  "top camera pass part zone"
  B3:7/9  "one shot"
  B3:7/10  "one shot"
  B3:7/11  "good part detected at top top"
  B3:7/12  "side camera pass part zone"
  B3:7/13  "one shot"
  B3:7/14  "passing part present bottom top camera"
  B3:7/15  "force boxing enable enables box tog bypass box plug in"
  B3:8/0  "bypass extra trigger camera 1"
  B3:8/1  "bypass extra trigger camera 2"
  B3:8/2  "bypass extra trigger camera 3"
  B3:8/3  "bypass extra trigger camera 4"
  B3:8/6  "a bypass bit"
  B3:8/7  "a bypass bit"
  B3:8/8  ET1_OLD  "extra trigger camera 1"
  B3:8/9  ET2_OLD  "extra trigger camera 2"
  B3:8/10  ET3  "extra trigger camera 3"
  B3:8/11  ET4  "extra trigger camera 4"
  B3:8/12  "start bottom top camera responce"
  B3:8/13  "extra blow signal for testing"
  B3:8/15  "start side camera responce"
  B3:9/2  "one shot"
  B3:9/4  "start top camera responce"
  B3:9/6  "C1D"
  B3:9/7  "C1t"
  B3:9/8  "C2D"
  B3:9/9  "C2t"
  B3:9/10  TEST_I1
  B3:9/11  I1_PASS_ZONE
  B3:9/12  I1_TRIG_TM_OK
  B3:9/14  "input from hmi to reset count"
  B3:10/0  "bypass part too close"
  B3:10/1  STRETCHED_BOX_IN_POS  "pulst stretch box in position sensor signal"
  B3:10/2  "One Shot"
  B3:10/3  "One Shot"
  B3:10/4  "changing Box chute door operation"
  B3:10/5  "one shot"
  B3:10/6  "excessive data output time"
  B3:10/9  "one shot"
  B3:10/10  "one shot"
  B3:10/11  "bottom part present trailling edge"
  B3:10/13  "one shot"
  B3:10/14  "Dont use"
  B3:10/15  "Reserved For Shift Registers"
  B3:11/0  "bypass unused portion of code"
  B3:11/1  "bypass"
  B3:11/2  "Enable encoder belt movement simulation when testing"
  B3:11/3  "Block blow signals while changing box"
  B3:11/4  "one shot"
  B3:11/6  "one shot"
  B3:11/7  "one shot"
  B3:11/8  "one shot"
  B3:11/11  "one shot"
  B3:11/12  "one shot"
  B3:11/13  TEST_TRIG_SIG
  B3:11/14  SOC  "start delay to false optic cycle"
  B3:11/15  "one shot"
  B3:12/0  "one shot"
  B3:12/1  "one shot"
  B3:12/2  "Command 2 Oneshot"
  B3:12/3  "Command 2 Active"
  B3:12/4  "Command3 Oneshot"
  B3:12/5  "Command 3 Active"
  B3:12/6  "Inspection Command Counter"
  B3:12/7  "Command 4 Active"
  B3:12/8  "Command 4 Oneshot"
  B3:12/14  "flip flop bit"
  B3:13/4  I3_PASS_OS
  B3:13/5  "bypass"
  B3:13/6  "Off"
  B3:13/7  "On"
  B3:13/8  "On"
  B3:13/9  "Off"
  B3:13/10  "On"
  B3:13/11  "Off"
  B3:13/12  "Test Trigger to laser Spacing"
  B3:13/15  "Test Signals"
  B3:17/12  "Always Off"
  B9:0/0  "Trigger Insert Position"
  B9:0/1  "bottom of top conveyor part transfer location"
  B9:0/[N7:0]  "Side Camera Trigger Posistion"
  B9:0/[N7:2]  "Mask Start Position"
  B9:0/[N7:6]  "Blow Off Position"
  B9:0/[N7:20]  "part present bit shift load position"
  B9:0/[N7:48]  "Top Camera Trigger Posistion"
  B9:0/[N16:0]  "Trigger Position"
  B9:0/[N17:8]  "part from bottom belt present at top belt optic position"
  B10:0/0  "Pass Insert Position"
  B10:0/1  TOP_CAM_LOAD
  B10:0/[N7:2]  "Pass Bit Position"
  B10:0/[N7:4]  "Pass Insert Position"
  B10:0/[N7:5]  "Pass Start Position"
  B10:0/[N7:6]  "Pass Position"
  B10:0/[N7:48]  TOPCAMTRIGPOS
  B10:0/[N16:4]  "Pass Insert Position"
  B10:0/[N16:6]  "Pass Position"
  B11:0/0  "Trigger Insert Position"
  B11:0/[N7:8]  "Fail Bit Position"
  B11:0/[N16:0]  "Trigger Position"
  B12:1/0  "Conveyor Start Oneshot"
  B12:1/1  "Feed Start Oneshot"
  B12:1/2  "Conveyor Stop Oneshot"
  B12:1/3  "Feed Stop Oneshot"
  B12:1/5  "Conveyor Start Oneshot"
  B12:2/8  BOXING  "BOXING System Wiring Is Connected"
  B12:2/10  OSR_42
  B12:2/11  BOX_IN_POS_OS  "BOXING Empty Box In Position One-Shot"
  B12:2/12  BOX_INDEXING  "BOXING Conveyor Indexing"
  B12:2/13  OSR_45
  B12:2/14  BOX_PLC_COUNTER  "BOXING PLC Counter Active Bit"
  B14:0/0  "Bottom Pass Insert"
  B14:0/4  "Bottom Pass Insert Position"
  B14:0/[N13:14]  "Start Laser Pass"
  B14:0/[N16:4]  "Pass Insert Position"
  B14:0/[N16:6]  "Pass Position"
  B15:0  "Alarm Bits"
  B18:1/1  "bottom pass one shot transfer"
  B18:3/2  "Part Present Oneshot"
  B18:3/3  "Part Present Oneshot"
  B18:5/11  "Transfer bottom pass result from end of bottom conveyor"
  B18:10/15  "Reserved For Shift Registers"
  B18:142  "fack camerea pass signal"
  B22:0  "Transfer Shift Register"
  B22:0/0  "load top conveyor bitshift from bottom cammera pass."
  B22:0/[N17:8]  "bottom good part at top optic position"
  B23:0/[N7:0]  "Bottom Pass Output"
  B25:0/4  UNUSED_4  "Unused Camera #4 Trigger"
  B189:0/10  TURN_OFF_BELT
  B191:0  MAJOR_ERROR
  B191:1  MINOR_ERROR
  B191:1/2  "Boxing conveyor backed up"
  B191:2  FLAG
  B202:0/8  AT_LOCATION_1_1
  B202:0/11  AT_LOCATION_2_1
  BOTTOM_CONVEYOR  
  C5:2  "Fault Counter"
  C5:5  "Trigger Count"
  C5:6  "Trigger Counter"
  C5:7  "Complete Counter"
  C5:8  BOX_CNT_1  "BOXING Quantity Counter #1"
  C5:9  BOX_CNT_2  "BOXING Quantity Counter #1"
  CHUTE_OPC  
  F8:0  "Fail Percent Raw"
  F8:4  BOT_OPTIC_CON_FAILS  "non pass optic"
  F8:5  "bottom top camera pass count"
  F8:6  "top top camera missed count"
  F8:7  "top side camera missed count"
  F8:8  "bot top camera missed part count"
  F8:11  AIR_MULTIPLIER_PSI  "main air multiplyer (PSI) old machine 0.093"
  F8:13  "error top"
  F8:15  "error bottom"
  F8:18  TOP_SPEED  "top belt speed average in pulses per second 290 Max; Verify"
  F8:20  "bot belt speed average in pulses per second"
  F8:21  BLOW_COMP_TIME
  F8:24  I2_SIDE_CON_FAILS  "auto stop non pass count side"
  F8:26  "Part bits loaded into BitShift"
  F8:27  MAX_TIME
  F8:28  "momentary rate in ppm"
  F8:29  "Count of signals passed to the blow valve"
  F8:30  BOT_NON_PASS_OLD  "Parts missed bot camera"
  F8:31  "Count of off alignment between top and bottom ALIGN_FAILS"
  F8:32  TIME_WINDOW
  F8:33  TOP_NON_PASS_OLD  "parts missed top camera"
  F8:34  "count of blow signals"
  F8:35  "rate difference"
  F8:36  2MIN_OF_RATE  "OLD AND NEW ADDED TOGETHER"
  F8:37  SQU_ERR
  F8:38  "averaged rate"
  F8:39  SIDE_NON_PASS_OLD  "parts missed side camera"
  F8:40  "absoloute difference top"
  F8:41  "absoloute difference bottom"
  F8:42  "Total fail and missed count CAM_NON_PASS"
  F8:43  "change in part rate as %"
  F8:44  "difference as a ratio of the total"
  F8:45  "TOO_CLOSE_BOT"
  F8:46  "TOO_WIDE_BOT"
  F8:48  "transfer"
  F8:49  "TOO_CLOSE_TOP"
  F8:50  I3_TOP_CON_FAILS  "auto stop non pass count top"
  F8:51  "TOO_WIDE_TOP"
  F8:52  "OPTO_FAILS"
  F8:53  "optic fail count top camera TOP_OPT_FAIL_CT"
  F8:54  "optic fail count bot camera BOT_OPT_FAIL_CT"
  F8:59  TOP_OPTIC_CON_FAILS  "non pass optic"
  F19:0  BOT_HS_COUNTER  "Bottom Encoder High Speed Counter"
  F19:4  "Conveyor Input Blip Counter"
  F188:1  "HMI Recerk speed input"
  F188:2  "HMI input for feed wheel speed"
  F188:3  "HMI input for feeder speed"
  F188:4  "HMI input for hopper speed"
  F192:0  "temp"
  HSC:0.3/6  "Underflow interrupt"
  HSC:0.3/7  "Overflow interrupt"
  HSC:1.3/6  "Underflow interrupt"
  HSC:1.3/7  "Overflow interrupt"
  I:0.0/0  "Encoder Signal "A""
  I:0.0/1  "Encoder Signal "B""
  I:0.0/3  "spare"
  I:0.0/7  INS_2_NOERR  "signal to indicate the inspection has completed without error or pass signal"
  I:0.0/8  INS_3_PASS
  I:0.0/9  INS_3_NOERR  "signal to indicate the inspection has completed without error or pass signal"
  I:0.0/10  INS_4_PASS
  I:0.0/11  INS_4_NOERR  "signal to indicate the inspection has completed without error or pass signal"
  I:0.0/12  INS_ERR  "cause the isnpection process to stop when overloaded Heart Beat"
  I:0.0/15  "Front E-Stop Active"
  I:0.1/0  "Rear E-Stop Active"
  I:0.1/1  "Front Door Open Switch Active On When Closed"
  I:0.1/2  "Rear Door Open Switch Active On When Closed"
  I:0.1/3  OVERRIDE  "Maintenance Mode Key Switch"
  I:0.2/3  "Packaging Conveyor full"
  I:0.2/4  "Packaging Conveyor Box in Position"
  I:0.4  "Spare Analog Input 1"
  I:0.5  "Spare Analog Input 2"
  I:0.6  "Spare Analog Input 3"
  I:2.0/2  BOX_PLUG_IN  "box connected input signal"
  I:2.0/3  PACK_HIGH  "Box Discharge Backed Up also cust fault"
  I:2.0/4  BOX_NOT_IN_POS  "and close door signal from cust boxing"
  L13:0  "multiplyer to translate percent"
  L13:1  "Last Part Count in Rate loop used to calculate the last cycle part count"
  L13:2  TOTAL_CAM_FAILS
  L13:3  "Part of Cam Fail Count Calculation"
  L13:4  "this Time Stamp"
  L13:5  VIRT_TMR_BLOW  "blow timer count in ms"
  L13:6  VIRT_TMR_BLOW2CHUTE  "count of time in ms for the blow to chute time"
  L13:7  MAX_FAIL_PERC_X_100
  L13:11  "Previous part time stamp"
  L13:15  "time since last part"
  L13:16  TRUE  "ONE TIME ENABLE FOR THE TIMES WHEN WE FORGET TO RE-ENABLE AFTER SHIPMENT"
  L13:17  FALSE
  L13:20  "last part to part time 10us"
  L13:21  "Max Value"
  L13:23  "missed count"
  L13:24  "missed count"
  L13:29  "missed count"
  L13:31  "do not use"
  L13:32  "do not use"
  L13:42  "i3 pass signal maximum on time"
  L13:44  "i3 pass signal maximum off time"
  L13:47  "Bot skip count"
  L13:48  "Side skip count"
  L13:49  "Top skip count"
  L14:0  TESTING_ENABLED
  L14:2  REAR_EMERG_STOP_OLD
  L14:3  FRONT_EMERG_STOP_OLD
  L14:4  REAR_DOOR_SW_OLD
  L14:5  FRONT_DOOR_SW_OLD
  L14:6  FEED_STATUS_OLD
  L14:7  CONVEYOR_STATUS_OLD
  L14:8  POWER_STATUS_OLD
  L14:9  BOX_JAM_FAULT_OLD
  L14:10  NO_BOX_FAULT_OLD
  L14:11  DSCRG_BACKUP_FAULT
  L14:12  MACHINE_FAULT_OLD
  L14:13  CNTER_SEOR_FLT
  L14:14  TOP_CONVEY_FLT_OLD
  L14:15  DN_TRACK_BLOD_FLT
  L14:16  AIR_PRESSURE_FAULT_O
  L14:17  AIR_PRESSURE_OLD
  L14:18  AIR_PRESSUREB
  L14:19  CURRENT_BOX_COUNT
  L14:20  CURRENT_BOX_COUNTB
  L14:21  PASSING_PART_COUNT
  L14:22  PASSING_PART_COUNTB
  L14:24  FAILING_PART_COUNTB
  L14:25  RATE
  L14:26  RATEB
  L14:27  RATE_DROP
  L14:28  RATE_DROPB
  L14:29  NON_PASS_BOT
  L14:30  NON_PASS_BOTB
  L14:31  NON_PASS_SIDE
  L14:32  NON_PASS_SIDEB
  L14:33  NON_PASS_TOP
  L14:34  NON_PASS_TOPB
  L14:35  CAM_NON_PASS
  L14:36  CAM_NON_PASSB
  L14:37  TOP_OPT_FAIL_CT_OLD
  L14:38  TOP_OPT_FAIL_CTB
  L14:39  BOT_OPT_FAIL_CT_OLD
  L14:40  BOT_OPT_FAIL_CTB
  L14:41  OPTO_FAILS
  L14:42  OPTO_FAILSB
  L14:43  TOO_CLOSE_BOT_OLD
  L14:44  TOO_CLOSE_BOTB
  L14:45  TOO_WIDE_BOT_OLD
  L14:46  TOO_WIDE_BOTB
  L14:47  ALIGN_FAILS_OLD
  L14:48  ALIGN_FAILSB
  L14:49  TOO_CLOSE_TOP_OLD
  L14:50  TOO_CLOSE_TOPB
  L14:51  TOO_WIDE_TOP_OLD
  L14:52  TOO_WIDE_TOPB
  L14:53  I1_REJECTS_FLT
  L14:54  FEED_WHEEL_STATUS
  L14:55  I2_REJECTS_FLT
  L14:56  I3_REJECTS_FLT
  L14:57  TOP_OP_REJECTS_FLT_O
  L14:58  BOT_CONVEY_FLT_OLD
  L14:59  BOTTOTOPALIGNMENT_OL  "Measurement of last offset of part alignment for part tracking between bottom system & top"
  L14:60  BOTTOTOPALIGNMENTB  "Measurement of last offset of part alignment for part tracking between bottom system & top"
  L14:61  TOP_BELT_SPEED_OLD  "Top Belt Speed x 1000"
  L14:62  TOP_BELT_SPEEDB  "Top Belt Speed B x 1000"
  L14:63  BOT_BELT_SPEED_OLD  "Bot Belt Speed x 1000"
  L14:64  BOT_BELT_SPEEDB  "Bot Belt Speed B x 1000"
  L14:65  BULK_DONE
  L15:0  MAX_PART_WIDTH_BOT_O
  L15:1  NU1
  L15:2  BOT_CAM_TRIG_POS
  L15:3  BOT_CAM_TRIG_POSB
  L15:4  BOT_TRANS_POINT_OLD
  L15:5  BOT_TRANS_POINTB
  L15:6  TRANS_ZONE_WIDTH_OLD
  L15:7  TRANS_ZONE_WIDTHB
  L15:8  TOP_OPTIC_POS_OLD
  L15:9  TOP_OPTIC_POSB
  L15:10  MAX_PART_WIDTH_TOP_O
  L15:11  MAX_PART_WIDTHB
  L15:12  MIN_PART_GAP_TOP_OLD
  L15:13  MIN_PART_GAP_TOPB
  L15:14  SIDE_CAM_TRIG_POS_OL
  L15:15  SIDE_CAM_TRIG_POSB
  L15:16  EXTRA_TRIG_POS
  L15:17  EXTRA_TRIG_POSB
  L15:18  TOP_CAM_TRIG_POS
  L15:19  TOP_CAM_TRIG_POSB
  L15:20  BLOW_OFF_POSITION_OL
  L15:21  BLOW_OFF_POSITIONB
  L15:22  MAX_CONT_REJECT
  L15:23  MAX_CONT_REJECTB
  L15:24  TOP_LOAD_POSITION_OL
  L15:25  TOP_LOAD_POSITIONB
  L15:26  BLOW_TIME_OLD
  L15:27  BLOW_TIMEB
  L15:28  BOT_CONV_SPEED_OLD
  L15:29  BOT_CONV_SPEEDB
  L15:30  TOP_CONV_SPEED_OLD
  L15:31  TOP_CONV_SPEEDB
  L15:32  BOX_COUNT_LIMIT_OLD
  L15:33  BOX_COUNT_LIMITB
  L15:34  BOT_OPTIC_LOC_OLD
  L15:35  BOT_OPTIC_LOCB
  L15:36  MIN_PART_GAP_BOT_OLD
  L15:37  MIN_PART_GAP_BOTB
  L15:38  FEEDER_SPEED_OLD  "15% min"
  L15:39  FEEDER_SPEEDB  "15% min"
  L15:40  HOPPER_SPEED_OLD  "15% min"
  L15:41  HOPPER_SPEEDB  "15% min"
  L15:42  ENABLE_BOXING_OLD
  L15:43  RESET_PLC_FAULT_OLD
  L15:44  ALIGNMENT_TRIGGERS_O
  L15:45  ENABLE_AIR_FAULT_OLD
  L15:46  TURN_OFF_CON_OLD  "HMI Stop Conveyors Push Button"
  L15:47  TURN_ON_CONVEYORS_OL  "HMI Start Conveyors Push Button"
  L15:48  TURN_OFF_FEEDER_OLD  "HMI Stop Feeder Push Button"
  L15:49  TURN_ON_FEEDER_OLD  "HMI Start Feeder Push Button"
  L15:50  RESET_ALL_COUNT_OLD
  L15:51  FORCE_PLC_FAULT
  L15:52  ENABLE_INSPECTION1
  L15:53  ENABLE_INSPECTION2_O
  L15:54  ENABLE_INSPECTION3
  L15:55  ENABLE_INSPECTION4
  L15:56  VISION_MAX_RES_MS_OL
  L15:57  VISION_MAX_RES_MSB
  L15:58  VISION_MIN_RES_MS
  L15:59  VISION_MIN_RES_MSB
  L15:60  RESET_FAIL_COUNT_OLD
  L15:61  RESET_BOX_COUNT_OLD  "HMI Box count Reset"
  L15:62  FEED_WHEEL_START
  L15:63  FEED_WHEEL_STOP
  L15:64  FEED_WHEEL_SPEEDOLD
  L15:65  FEED_WHEEL_SPEEDB
  L15:66  MAX_BLOW2CHUTE_MS_OL
  L15:67  MAX_BLOW2CHUTE_MSB
  L15:68  BULK_ENABLE
  L23:0  POWER_ON
  L23:1  MPCE_ON
  L23:2  FRONT_ESTOP_ON
  L23:3  REAR_ESTOP_ON
  L23:4  MSCE_ON
  L23:5  FRONT_DOOR_CLOSED
  L23:6  REAR_DOOR_CLOSED
  L23:8  MAINTENANCE_DUE
  L23:9  CONVEYOR_ON
  L23:10  FEED_ON
  L23:11  BOT_OPT_FAIL_CT
  L23:12  BOT_NON_PASS  "parts missed BOT camera"
  L23:13  BOT2TOP_ALIGNMENT
  L23:14  ALIGN_FAIL_CT
  L23:15  TOO_CLOSE_TOP
  L23:16  TOP_TOO_WIDE
  L23:17  TOO_CLOSE_BOT
  L23:18  TOO_WIDE_BOT
  L23:19  TOP_OPT_FAIL_CT
  L23:20  TOTAL_OPTIC_FAILS
  L23:21  BOT_OP_CON_FAILS_FLT
  L23:22  I2_CON_FAILS_FLT
  L23:23  TOP_OP_CON_FAILS_FLT
  L23:24  I3_CON_FAILS_FLT
  L23:25  I1_CON_FAILS_FLT
  L23:26  LAST_BOT_OFFSET  "Last part offset since pass from trigger location for setup evaluation"
  L23:27  LAST_SIDE_OFFSET  "Last part offset since pass from trigger location for setup evaluation"
  L23:28  LAST_TOP_OFFSET  "Last part offset since pass from trigger location for setup evaluation"
  L23:29  SIDE_NON_PASS  "parts missed side camera"
  L23:30  TOP_NON_PASS  "Parts Missed Top Camera"
  L23:31  BLOW2CHUTE_TIME
  L23:32  ANY_FAULT
  L23:33  PAK_DSC_BACKUP_FAULT
  L23:34  AIR_PRESSURE_FAULT
  L23:35  DN_TRACK_BLOCKED_FLT
  L23:36  COUNTER_SESOR_FAULT
  L23:37  BOX_JAM_FAULT
  L23:38  TOP_CONVEY_FLT
  L23:39  BOT_CONVEY_FLT
  L23:40  TOP_SPEED_OUTPUT
  L23:41  BOT_SPEED_OUTPUT
  L23:42  TOP_SP_ACT_X1000
  L23:43  BOT_SP_ACT_X1000
  L23:45  BLOW_COUNT
  L23:46  RATE_CHANGE
  L23:47  CHUTE_OPTIC_COUNT
  L23:48  RATE_LAST_PPM
  L23:49  AVERAGED_RATE  "parts per minute"
  L23:50  BOX_COUNT
  L23:51  BOXING_ON
  L23:52  NO_BOX_FAULT
  L23:53  TOTAL_FAIL_COUNT
  L23:54  MAXRATEDROP_FAULT
  L23:55  PERCENTFAIL_X100
  L23:56  TOTAL_COUNT
  L23:57  FAIL_PERCENT_FAULT
  L23:58  BOT_RES_WIDTH
  L23:59  SIDE_RES_WIDTH
  L23:60  TOP_RES_WIDTH
  L23:61  BULK_BOXING
  L23:62  CUST_BOXING
  L23:63  BULK_CT_REACHED_FLT
  L24:0  EI1  "Enable Inspection 1"
  L24:1  I1_BOT_TRIG_LOC
  L24:2  EET1  "ENABLE EXTRA TRIGGER"
  L24:3  ET1_DELAY
  L24:4  HMI_RESET_FLT_BUTTON
  L24:5  ENABLE_BOXING
  L24:6  TURN_OFF_CONVEYORS
  L24:7  TURN_ON_CONVEYORS
  L24:8  TURN_OFF_FEEDER
  L24:9  TURN_ON_FEEDER
  L24:10  FEEDER_SPEED
  L24:11  FEED_WHEEL_SPEED
  L24:12  HOPPER_SPEED
  L24:13  BOT_OPTIC_LOC
  L24:14  MAX_PART_WIDTH_BOT
  L24:15  BOT_TRANS_LOC
  L24:16  TOP_OPTIC_LOC
  L24:17  TOP_LOAD_LOC
  L24:18  TRANS_ZONE_WIDTH
  L24:19  MIN_PART_GAP_TOP
  L24:20  MAX_PART_WIDTH_TOP
  L24:21  EN_ALIGN_TRIG
  L24:22  I2_SIDE_TRIG_LOC
  L24:23  EI2  "Enable Inspection 2"
  L24:24  EET2  "ENABLE EXTRA TRIGGER"
  L24:25  ET2_DELAY
  L24:26  I3_TOP_TRIG_LOC
  L24:27  EI3  "Enable Inspection 3"
  L24:28  EET3  "ENABLE EXTRA TRIGGER"
  L24:29  ET3_DELAY
  L24:30  BLOW_OFF_LOC
  L24:31  BLOW_TIME
  L24:32  MAX_CON_FAILS
  L24:33  ENABLE_AIR_FAULT
  L24:34  MIN_AIR_PRESSURE
  L24:35  GD_PT_SEN_BLKED_TM
  L24:36  EN_CT_BL_TM_FAULT  "ENABLE THE COUNTER SENSOR FAULT BASED ON BLOCKED TIME"
  L24:37  MAX_BLOW2CHUTE_MS
  L24:38  EN_CH_FLT_NO_BLOW
  L24:39  TOP_CONV_SETTING
  L24:40  BOT_CONV_SETTING
  L24:41  BOX_COUNT_LIMIT
  L24:42  RESET_ALL_COUNT
  L24:43  RESET_FAIL_COUNT
  L24:44  MIN_PART_GAP_BOT
  L24:45  VISION_MAX_RES_TIME
  L24:46  VISION_MIN_RES_TIME
  L24:47  RESET_BOX_COUNT  "HMI Reset Box Count"
  L24:48  BOXING_OPTION
  L24:49  SUDO
  L24:50  MAXDROP
  L24:52  MAX_FAIL_PERCENT
  L24:53  SETUP_REQUEST
  L24:54  MAX_SETUP_TIME
  L24:55  MAX_STOPPED_TIME
  L42:51  CHUTE_STABLIZING
  L100:0  MINOR
  L100:1  MAJOR
  L187:0  ALIGN_OFFSET_MIN
  L204:3  "temp count for HMI heartbeat"
  N7:0  SIDE_TRIG_POS_INTEGE  "Side Trigger Position"
  N7:1  "sudo part interval"
  N7:2  "Min Part Spacing top"
  N7:4  "distance from last trigger"
  N7:5  "top part too close or too wide or not aligned distance measurement"
  N7:6  BLOW_LOC_INTEGER  "Blow-off Position"
  N7:7  "Top Conv Speed"
  N7:8  "Bottom Conveyor Speed"
  N7:9  "Minimum Spacing measurement"
  N7:10  BOT_PART_LOAD_PT
  N7:11  "1/2 bottom optic part width"
  N7:12  "second side trigger position"
  N7:13  SIDE_TEST_OFFSET  "max distance from trigger to check for pass part signal"
  N7:14  BLOW_LOCATION2
  N7:15  "Second bottom trigger position"
  N7:16  "distance to add to optic position to remove part present locations for parts too close top"
  N7:17  TOP_PT_WIPE_LOC  "location to remove part present signals when signals are too close"
  N7:18  "total distance to remove part present signals when parts are too close top"
  N7:19  "sudo timer count"
  N7:20  "1/2 top optic part width"
  N7:21  BOT_TRIG_POS_INTEGER  "Trigger Position"
  N7:22  TOP_TEST_OFFSET  "max distance from trigger to check for pass part signal"
  N7:23  "part width as measured at top optic part present sensor"
  N7:24  TOP_PT_WIDTH_TEMP  "check part width temporty counting"
  N7:25  TM_WINDOW  "Interger Time Window"
  N7:27  "max part width top optic"
  N7:28  BOT_TRIG_POS_OLD  "Trigger Position"
  N7:29  "belt travel to wipe parts off of belt when fell part detected"
  N7:30  "tempory counting bit to measrue top belt speed"
  N7:31  TOP_PART_LOAD_PT
  N7:32  TOP_OPT_LOC  "Used As Indirect Address"
  N7:33  "pps top belt"
  N7:34  "belt travel since fell part detected"
  N7:35  "distance since bottom part passed signal at top optic"
  N7:36  TRANS_ZONE  "distance to allow for part shift when part travels from bottom belt to top optic"
  N7:37  "bottom optic part width"
  N7:38  "blow to optic time"
  N7:39  BOT_PT_WIDTH_TEMP  "check part width temporty counting"
  N7:40  BOT_TRANS_POS  "bottom conveyor pass signal transfer position"
  N7:41  "Maximum Time from blow Signal to Optic Chute Optic Crosing MAX_BLOW2CHUTE_MS"
  N7:42  "second top trigger position"
  N7:43  BLOW_OFFSET_LOCATION
  N7:44  LAST_BOT_OFFSET_R  "Last part offset since pass from trigger location for setup evaluation"
  N7:45  SIDE_TEST_WIDTH  "side pass zone width"
  N7:46  SIDE_SINCE_PASS  "distance since side camera pass"
  N7:47  SIDE_TEST_LOC  "Location of pass window"
  N7:48  TOP_TRIG_POS_INTEGER  "Top Trigger Position"
  N7:49  TOP_SINCE_PASS  "distance since top camera pass"
  N7:50  TOP_TEST_LOC  "Location of pass window"
  N7:51  "side camera response time ms"
  N7:52  "Part Rate as interger"
  N7:53  "bot belt speed as interger"
  N7:54  "side camera responce distance"
  N7:55  "top camera responce distance"
  N7:56  "top camera responce time ms"
  N7:58  BLOW_OFFSET
  N7:60  BOT_OPT_LOC  "bottom optic location"
  N7:61  "counting bit for distance since last part trigger for bottom"
  N7:62  "distance since last part trigger bottom"
  N7:63  "min part spacing bottom"
  N7:64  "bot part too close or too wide distance measurement"
  N7:65  "tempory counting bit to measrue bottom belt speed"
  N7:66  "pps bottom belt"
  N7:68  "total distance to remove part present signals when parts are too close bottom"
  N7:69  "distance to add to optic position to remove part present locations for parts too close bottom"
  N7:70  BEC  "bottom encoder count"
  N7:71  BOT_PT_WIPE_LOC  "location to remove part present signals when signals are too close"
  N7:72  "max part width bottom optic"
  N7:73  TEC  "top encoder count"
  N7:74  BOT_SINCE_PASS  "distance since bottom inspection 1 pass"
  N7:75  BOT_TEST_OFFSET  "max distance from trigger to check for pass part signal"
  N7:76  BOT_TEST_LOC  "Location of pass window."
  N7:77  BOT_TEST_WIDTH  "bot pass zone width"
  N7:79  "bottom top camera responce distance"
  N7:80  "bottom top camera responce time"
  N7:81  "bottom to top offset"
  N7:82  TOP_LOAD_LOCATION  "Used As Indirect Address"
  N7:83  "last part count for rate"
  N7:85  "measure movement"
  N7:86  "fake part optic far edge position to virtual real part"
  N7:100  2ED_BOT
  N7:101  3ED_BOT
  N7:102  2ED_SIDE
  N7:103  3ED_SIDE
  N7:104  2ED_TOP
  N7:105  3ED_TOP
  N7:121  "Deformed Head Blowoff Timer Preset (s)"
  N10:1  "old ConveyorStatus"
  N10:2  "PowerOn"
  N10:3  "Local Mode On BypassBoxingPLC"
  N10:4  "Boxing Connected Signal"
  N10:5  "BoxJamSignal"
  N10:6  "WaittingOnBoxSig"
  N10:7  "ConveyorFullSig"
  N10:8  "MachineFaultSig"
  N10:9  "Counter Sensor Fault"
  N10:11  "Feeder Track Sensor Blocked"
  N10:12  "Air Pressure Fault"
  N13:0  "Part Inspecting"
  N13:4  "Completed Counter"
  N13:5  "Trigger Position Counter"
  N13:6  "BlowOff Start Counter"
  N13:7  "BlowOff Stop Counter"
  N13:8  "Inspection Command Counter"
  N13:9  "Complete Counter"
  N13:10  "Pass Signal Counter"
  N13:11  "Solenoid Signal Counter"
  N13:12  "Hold Pass Counter"
  N13:13  "Hold Pass Length"
  N16:0  BOT_TRIGGER_OLD  "Trigger Position"
  N16:1  "Bottom Inspection Offset For Tracking"
  N16:3  "Bit Shift Preset"
  N17:5  "Parts In Tube Counter"
  N17:6  "Parts In Tube Limit"
  N17:9  "Bot to Top Transfer Position"
  N17:12  "Trigger to laser Counter"
  N186:0  LOAD_LOCATION
  N186:1  OPTIC_LOCATION
  N197:5  "Feeder Speed Output Setting"
  N197:10  "pulse distance to keep blow on then turn off feed"
  N197:11  "speed in pps"
  N197:12  "seconds of ontime"
  N200:25  T6POS1
  N203:7  ALIGNMENT_OFFSET  "difference between real and virtual part location"
  O:0.0/1  "spare"
  O:0.0/3  INS_2_TRIG
  O:0.0/4  INS_3_TRIG
  O:0.0/5  INS_4_TRIG
  O:0.0/9  "spare"
  O:0.0/10  "spare"
  O:0.0/11  "Spare"
  O:3.0/0  "Ready-Run signal to Boxer? Always on unless fault?"
  O:3.0/2  "Customers pecies counting done signal (Change Box?)"
  O:3.0/4  GRN_LT  "Green Light"
  O:3.0/5  AMB_LT  "Amber Light"
  O:3.0/6  RED_LT  "Red Light"
  O:3.0/7  "Spare"
  O:3.0/8  "spare"
  O:3.0/9  TOP_CNV_INHIBIT
  PFILE:6  "check for part jams"
  Q2:55  END_OF_MAIN
  Q5:94  END_OF_BELTS
  R6:5.POS  "Empty Fifo"
  R21:0  "Trigger Shift Register"
  T4:5  TOP_BELT_TMR2  "Fine Delay to test Top belt movement"
  T4:7  "Boxing conveyor full error delay"
  T4:8  PRO_SLOW_TMR  "How long has the rate been slow for"
  T4:9  "optio hold holds minimum optic time to 16ms"
  T4:10  BOT_BELT_TMR2  "Fine Delay to test Bot belt movement"
  T4:11  "belt stop delay timer"
  T4:12  "Hopper On Delay"
  T4:13  ETT1  "EXTRA TRIGGER TIMER"
  T4:14  ETT2  "EXTRA TRIGGER TIMER"
  T4:15  GOOD_PES_TMR  "Good Part Sensor Blocked Timer"
  T4:16  ETT3  "EXTRA TRIGGER TIMER"
  T4:17  "Stopped Time Out Timer"
  T4:18  BOX_JAM_FLT_TMR  "BOXING In Position Sensor Timer"
  T4:19  BOX_WAIT  "BOXING Waiting For Empty Box Timer"
  T4:20  BOX_EXIT_TMR  "BOXING Exit Conveyor Sensor Timer"
  T4:21  DN_TRACK_SENSOR_TMR  "Feeder Track Sensor Blocked Timer"
  T4:22  TOP_BELT_TMR  "Corse Delay to test Top belt movement"
  T4:23  "SETUP TIMER"
  T4:24  "bot cam responce timmer 2"
  T4:25  "box in posistion pulse stretcher timer"
  T4:27  "Timer to allow parts to pass through shoot"
  T4:28  "Timer to allow shoot door to close"
  T4:29  "Part Rate Timer"
  T4:30  "Hopper Off Delay"
  T4:31  BOT_BELT_TMR  "Corse Delay to test Bot belt movement"
  T20:0  "Trigger On Time"
  T23:0  T25
  U:5  "conveyor"
  U:9  "slow data"
  U:11  "transfered data calcuations from the high speed section"
  U:28  "faults"
  U:29  "speed"
  U:30  "count"
  U:31  "rate calc"
  U:32  "boxer"
  U:33  "bulk pack"
  U:34  "customer boxing unit signals"
  U:35  "cleanup"
  U:140  "inspection 6 trigger"
  U:141  "inspection 6 result"
  U:151  "inspection 7 result"

COMMENTS NOT ATTACHED TO A CURRENT RUNG
  N17:8: ****************************************************************************************************************
    I can not find anywhere in the program where the "Test Spacing From Pickup to Trigger is activated indicating to me that this entire function must not be doing anything in this program at this time.
    ****************************************************************************************************************
  T20:2: The timer used to verify that the part that triggered the top laser optic has passed the bottom camer. needs to be count
  T20:2.ACC: This rung is starting a timer that should be activated directly before the laser optic part presense sensor on the top conveyer and should cause the top optic to be ignored if the bottom camera system didn't pass. however other arrangements must be made if the bottom camera isn't going to be used as is the case with a nut inspection.
  B22:0/0: ***********************
     Bottom Part Syncronizing Logic
    ***********************
    
    This is the point at the bottom of the top conveyor where the part jumps from the bottom conveyor.  This system will then track the part through the top system to the point of the laser optic in order to verify that the part in question has passed the bottom inspection.  I believe that we NEED to include FAILING inspections to eliminate the possibility of a out of position part from passing. LW 072010
  C5:4: tempory counting to verify pass part count with boxing part count.
  N7:25: 1050
  B23:0/0: Yet another bit shift load with data in the part position indicating that there was a bottom system part pass as well as a top system part present at this location.
    
    verified works w/bypassed 071910 and unbypassed 072010
  I:0.0/8: special rung for testing. This rung can simulate a pass signal. It will not be timed correctly.
  F8:13: *************************
    Loads Side Camera Passing data into a bit shift
    *************************
    
    loads passing data bit into passing data bit shift register at the part present cl.
  B3:7/9: ************************************
     The next 3 rungs appear to do nothing
    ***********************************
  B11:0/0: load part present bit shit with one shot data from the part present sensor
  N7:45: not fully functional because of part overlap but measurems the camera responce time when part inspections are not overlaping
  F8:0: Counter inside of a high speed counter interrupt counts the number of Bit Shifts that need to be processed in order to move the logic with the parts on the conveyor.
  B3:6/1: ***********************
    Part Width and  Location
    ***********************
    
    Calculates the position of parts on the top belt by measureing the part width by calculating the number of belt movement pulses that occure when the optic is blocked and then devides that in half and add that to the optic location in the part presnet bit shift when the top optic is cleared.
  B3:6/0: make a bit come on indicating that a part that passed the bottom camera is within  range when crossing the top camera.
  B3:0/7: ********************
    Passing Part at Blow Position
    
    Blow signal is not retriggerable. If any signals are received prior to previous compleation of the blow process the signal will be ignored. Future changes may include tests or faults to verify that multiple blow signals are not overlaping.
    ********************
  B9:0/[N7:47]: Remove any part present signals outside of expected location
  O:0.0/3: **************
    Side Camera Trigger
    *************
  B9:0/[N7:50]: Remove any part present signals outside of expected location
  B3:4/14: *****
    Convertion of the optic signal to something stable
    *****
  F19:0: Counter inside of a high speed counter interrupt counts the number of Bit Shifts that need to be processed in order to move the logic with the parts on the conveyor.
  F8:14: **************
    Bottom Top Camera Trigger
    *************
    
    Trigger Bottom Top Camera
  B3:6/8: ********************************************************************************************************************************
    Box count reached
    Redo all of boxing;
    1. handle box done, change, box not moving, no new box
    2. everything else is situational, i.e. box removed, box not present
    add bulk pack rutine that just stops bowl and doesn't change box.
    ********************************************************************************************************************************
  N10:4: test if boxing is connected
  T4:27: Time to clear shoot
  T4:28: Time to close shoot door
  L13:2: Reset box count
  B3:11/3: After initial delay allow blow two start functioning
  B3:6/9: Detect fault condition no box present on conveyor
  L13:20: The following lines of code calculate the minimum and maximum time between evaluations. This is used for troubleshooting result timing issues.
  L14:5: on when ok to run, rear off turns both off
  L14:2: off when ok to run
  L14:3: off when ok to run
  L14:8: on when ok for run
  N7:76: removed relieance on trigger signal
  N197:20/0: Passes deformed head blowoff command to TOP PLC where solenoid output is located.
  N7:47: ***********************************************************************************************************************************************************
    From side
    ***********************************************************************************************************************************************************
    
    removed relieance on trigger signal
  O:0.0/4: **************
    Top Camera Trigger
    *************
  N7:50: ***********************************************************************************************************************************************************
    From top
    ***********************************************************************************************************************************************************
    
    removed relieance on trigger signal
  B3:10/1: prevents momentary signals from box present sensor from tripping the logic for box not present
    
    This is in responce to a problem created by the sensor occasionally turning on as if no box was in its path when there is a box present.
  B3:6/2: IF PROCESSING FAULT OCURES AT COUNTER SENSOR; CLEAR THE BELT OF PASSING DATA
  L14:36: ****************  nEEDS fIXING  **********************
  L14:23: ****************  nEEDS fIXING  **********************
  RUNG000012-000001: 1/2 of the transfer process. The other half is in the Top Optic file.
  RUNG000012-000000: 1/2 of the transfer process. The other half is in the Top Optic file.
  RUNG000010-000018: Remove any part present signals outside of expected location
  RUNG000010-000014: ****
                      Zeros out the non passing part count when one passes
    ****
  RUNG000010-000007: **************
    Bot Camera Trigger
    *************
  N7:46: Remove any part present signals outside of expected location

REVISION NOTES
  13: updated count reset
  14: added io moduals
  15: multiple steps toward new hmi integration
  21: test

DATA TABLE (non-zero values as saved)
DATA B3
% B3:0 % 0X6001 0X0002 0X0000 0X0626 0X0840 0X2400 0X02C0 0X0020 0X4007 0X0000
% B3:10 % 0X2041 0X0846 0X2000 0X0000
DATA T4
% .PRE .ACC %
% T4:0 % 300 304
% T4:1 % 150 0
% T4:2 % 32765 0
% T4:3 % 32765 0
% T4:4 % 32765 0
% T4:5 % 35 0
% T4:6 % 5555 5555
% T4:7 % 10 0
% T4:8 % 300 0
% T4:9 % 30 0
% T4:10 % 35 0
% T4:12 % 50 0
% T4:13 % 222 0
% T4:14 % 222 0
% T4:15 % 180 0
% T4:16 % 222 0
% T4:17 % 300 0
% T4:18 % 8 0
% T4:19 % 6 0
% T4:20 % 10 0
% T4:21 % 100 0
% T4:22 % 20 0
% T4:23 % 900 0
% T4:24 % 1000 0
% T4:25 % 250 250
% T4:26 % 666 666
% T4:27 % 400 0
% T4:28 % 400 0
% T4:29 % 10 0
% T4:30 % 50 50
% T4:31 % 20 0
% T4:32 % 69 0
DATA R6
% .LEN .POS %
% R6:0 % 4 0
% R6:1 % 4 0
% R6:2 % 2000 0
% R6:4 % 2048 0
% R6:5 % 2048 0
% R6:6 % 2048 0
% R6:7 % 2048 0
% R6:8 % 4 0
DATA N7
% N7:0 % 1226 46 30 0 4013 91 1466 101 101 32767
% N7:10 % 4 3 1227 0 1455 123 60 1090 90 17
% N7:20 % 4 122 0 7 0 30 -403 30 132 650
% N7:30 % 0 1034 1030 0 657 32767 18 5 0 0
% N7:40 % 1198 180 1237 1454 9 0 32767 1226 1236 32767
% N7:50 % 1236 0 175 16 0 0 0 1464 12 0
% N7:60 % 1 32767 4012 20 31 0 0 15 30 20
% N7:70 % 0 21 23 27738 32767 0 122 0 16 0
% N7:80 % 0 6 95 0 0 0 5 500 0 0
% N7:90 % 2011 4 4 12 1 0 0 0 0 1600
% N7:100 % 123 124 1227 1228 1237 1238 0 0 0 0
% N7:110 % 0 0 0 0 0 0 0 0 400 0
% N7:120 % 25007 61 0 0 0 0 0 0 0 0
DATA F8
% F8:0 % 17845.55 222 63265.63 0 0
% F8:5 % 0 0 0 0 112
% F8:10 % 0.0888 0.08897486 1263 101 63.26563
% F8:15 % 37.73437 4040 112 0 0
% F8:20 % 0 0.02 0 1 0
% F8:25 % 0 932781 0.222 279.6551 848597
% F8:30 % 0 170 0.03 38 852060
% F8:35 % 0 0 0 0 77
% F8:40 % 101 37.73437 0 100 1
% F8:45 % 1 2 0.21455 0 0
% F8:50 % 0 0 1 0 1
% F8:55 % 2000000 -221 0 0 0
% F8:95 % 0 0 0 25 0.00025
DATA B9
% B9:130 % 0X0000 0X0000 0X0000 0X0000 0X2000 0X0000 0X0000 0X0000 0X0000 0X8000
% B9:140 % 0X2480 0X0000 0X0000 0X0000 0X0000 0X0000 0X0000 0X0000 0X0000 0X0000
% B9:160 % 0X0000 0X0000 0X0000 0X0000 0X0000 0X0000 0X2000 0X0002 0X0000 0X0000
% B9:170 % 0X0000 0X0000 0X0000 0X2000 0X0000 0X0000 0X0000 0X0000 0X0000 0X0000
% B9:180 % 0X0000 0X0000 0X0000 0X0000 0X0000 0X0002 0X0000 0X0000 0X0000 0X0000
% B9:190 % 0X0010 0X0000 0X0000 0X0000 0X0000 0X0000 0X0000 0X0000 0X0000 0X0000
% B9:200 % 0X2B64 0X2B64 0X0000 0X0010 0X0000 0X2000 0X0000 0X0000 0X0000 0X0000
% B9:220 % 0X0000 0X0000 0X0000 0X0200 0X0000 0X0000 0X0000 0X0000 0X0000 0X0020
% B9:230 % 0X0040 0X0000 0X0000 0X0000 0X0000 0X0000 0X0000 0X0000 0X0000 0X0000
DATA B11
% B11:180 % 0X0000 0X8000 0X0000 0X0000 0X0000 0X0000 0X0000 0X0000 0X0000 0X0000
% B11:240 % 0X0000 0X0000 0X0000 0X4000 0X0000 0X0000 0X0000 0X0000 0X0000 0X0000
DATA L13
% L13:0 % 10000 0 17 17 -958747195
% L13:5 % 40 350 1000000 371112247 371112270
% L13:10 % 23 -1767500687 656931333 3364690 3364678
% L13:15 % 808753492 65535 -65536 2147483647 282
% L13:20 % 511654 808755107 653563960 17 0
% L13:25 % 25 -1428297619 -1767500734 339203115 0
% L13:30 % 280 200000 500000 85 132
% L13:35 % 217 217 217 15 25
% L13:40 % 15 0 28 3364544 0
% L13:50 % 18974 2147483647 2147483647 0 0
DATA L23
% L23:0 % 65535 -65536 -65536 -65536 -65536
% L23:5 % -65536 -65536 112 65535 -65536
% L23:10 % -65536 0 17 10 17
% L23:15 % 0 0 0 0 8
% L23:20 % 0 -65536 -65536 -65536 -65536
% L23:25 % -65536 20 19 20 0
% L23:30 % 0 0 -65536 -65536 -65536
% L23:35 % -65536 -65536 -65536 -65536 -65536
% L23:40 % 16270 18414 0 63266 -65536
% L23:45 % 5062 0 0 0 0
% L23:50 % 0 -65536 -65536 17 -65536
% L23:55 % 33 5079 -65536 0 0
% L23:60 % 0 -65536 -65536 -65536 0
DATA L24
% L24:0 % -65536 122 -65536 222 -65536
% L24:5 % 65535 -65536 -65536 -65536 -65536
% L24:10 % 50 27 0 1 23
% L24:15 % 1198 1030 95 18 30
% L24:20 % 30 -65536 1226 -65536 -65536
% L24:25 % 222 1236 -65536 -65536 222
% L24:30 % 1466 27 10000 -65536 55
% L24:35 % 180 -65536 180 65535 101
% L24:40 % 101 1000 -65536 -65536 10
% L24:45 % 222 192 -65536 0 -65536
% L24:50 % -999 30 10000 65535 900
DATA L42
% L42:0 % -65536 0 0 0 0
% L42:5 % 45 45 45 0 0
% L42:20 % 0 0 32766 32766 0
% L42:50 % 0 30
DATA L183
% L183:0 % 50 216325420 12 1000000000 0
% L183:5 % 156634425 0 111 0 0
DATA N184
% N184:0 % 100 0 0 0 0 0 0 0 0 0
DATA B185
% B185:0 % 0X8000 0X0081 0X0000 0X0000 0X0000 0X0000 0X0000 0X0000 0X0000 0X0000
DATA N186
% N186:0 % 100 0 0 0 0 0 0 0 0 0
DATA L187
% L187:0 % 0 5 0 0 0
% L187:5 % 1062 4 1070 0 0
DATA F188
% F188:0 % 6 66 11 44 29
DATA B189
% B189:0 % 0X01F0 0X0000 0X0000 0X0000 0X0000 0X0000 0X0000 0X0000 0X0000 0X0000
DATA L190
% L190:0 % 0 5 0 0 1
% L190:5 % 0 0 0 1066 4
% L190:10 % 1070 0 1 0 0
DATA L192
% L192:0 % 371245004 371245004 1692 23 38422
% L192:5 % 100000 3000000 19 1 19
% L192:10 % 1 19 19 16 17
% L192:15 % 20 20 21 21 210
% L192:20 % 180 0 0 0 0
DATA F193
% F193:0 % 59.90296 0.315 0.022 6 60
% F193:5 % 0.09704208 0.015 0.001455631 7.0931 232.4125
% F193:10 % 0.011 0.195 0.165 0.337 0.348
% F193:15 % 210 180 0 0 0
DATA B196
% B196:0 % 0X00D5 0X180E 0X0905 0X0000 0X0000 0X0000 0X0000 0X0000 0X0000 0X0000
% B196:30 % 0X0000 0X0000 0X0001 0X0000 0X0000 0X0000 0X0000 0X0000 0X0000 0X0000
DATA N197
% N197:0 % 0 222 1111 2500 2500 14417 5555 300 150 0
% N197:10 % 4000 969 4 0 0 0 0 0 0 0
% N197:30 % 13 48 0 0 0 0 0 0 0 0
DATA B198
% B198:0 % 0X0009 0X0000 0X0000 0X0000 0X0000 0X0000 0X0000 0X0000 0X0000 0X0000
DATA L199
% L199:0 % 0 728209 134 11 6
% L199:5 % 5 5 5 5 174972
% L199:10 % 0 155 15 49 0
% L199:15 % 11877125 64440373 64441194 67620565 51
% L199:20 % 11877151 0 0 0 0
DATA N200
% N200:0 % 3 115 1 4 1321 145 333 444 555 0
% N200:10 % 2560 2560 2560 2560 146 2560 0 0 0 0
DATA L201
% L201:0 % 47 15 0 -3011735 44
% L201:5 % 11877319 0 0 -3010662 0
% L201:10 % 0 0 0 327 43
% L201:15 % 0 43 0 43 36830
DATA B202
% B202:0 % 0X0240 0X0000 0X0000 0X0000 0X0000 0X0000 0X0000 0X0000 0X0000 0X0000
DATA N203
% N203:0 % 135 136 136 353 354 354 464 0 465 465
% N203:10 % 575 576 576 0 0 0 0 0 0 0
DATA L204
% L204:0 % 555 100 5000 63962 3061
% L204:5 % 2501 2500 4000 0 0
DATA F205
% F205:0 % 9829.8 23591.52 14744.7 19659.6 0
